END_VAR
VAR CONSTANT
	(* prefix to unify the test names *)
	TEST_NAME_PREFIX		:STRING := 'assert.dateAndTime.simple.dateAndTime.';
	(* max value of a DWORD *)
	{attribute 'hide'}
	MAX_DWORD				:DWORD := 16#FFFF_FFFF;
	(* min value of a DWORD *)
	{attribute 'hide'}
	MIN_DWORD				:DWORD := 16#0000_0000;
	(* only the msb is set *)
	{attribute 'hide'}
	MSB_ONLY				:DWORD := 16#8000_0000;
	(* only the msb is set *)
	{attribute 'hide'}
	LSB_ONLY				:DWORD := 16#0000_0001;
	(* all bits set except the msb *)
	{attribute 'hide'}
	WITHOUT_MSB 			:DWORD := 16#7FFF_FFFF;
	(* for every nibble is the msb set only *)
	{attribute 'hide'}
	ALL_NIBBLE_MSB			:DWORD := 16#8888_8888;
	(* for every nibble is the msb unset only *)
	{attribute 'hide'}
	WITHOUT_NIBBLE_MSB		:DWORD := 16#7777_7777;
	(* for every nibble is the lsb set only *)
	{attribute 'hide'}
	ALL_NIBBLE_LSB			:DWORD := 16#1111_1111;
	(* every bit is set except the lsb *)
	{attribute 'hide'}
	LSB_IS_UNSET			:DWORD := 16#FFFF_FFFE;
	(* max vale of date and time *)
	DT_MAX					:DT := TO_DT(MAX_DWORD);
	(* min vale of date and time *)
	DT_MIN					:DT := TO_DT(MIN_DWORD);
	(* only the msb is set *)
	DT_MSB_ONLY				:DT := TO_DT(MSB_ONLY);
	(* all bits set except the msb *)
	DT_WITHOUT_MSB 			:DT := TO_DT(WITHOUT_MSB);
	(* for every nibble is the msb set only *)
	DT_ALL_NIBBLE_MSB		:DT := TO_DT(ALL_NIBBLE_MSB);
	(* for every nibble is the msb unset only *)
	DT_WITHOUT_NIBBLE_MSB	:DT := TO_DT(WITHOUT_NIBBLE_MSB);
	(* for every nibble is the lsb set only *)
	DT_ALL_NIBBLE_LSB		:DT := TO_DT(ALL_NIBBLE_LSB);	
	(* every bit is set except the lsb *)
	DT_LSB_IS_UNSET			:DT := TO_DT(LSB_IS_UNSET);
	(* only the msb is set *)
	DT_LSB_ONLY				:DT := TO_DT(LSB_ONLY);
END_VAR

THIS^.runValueIsEqualToTests();
THIS^.runValueIsGreaterThanTests();
THIS^.runValueIsInRangeOfTests();
THIS^.runValueIsLessThanTests();
THIS^.runValueIsMaxTests();
THIS^.runValueIsMinTests();
THIS^.runValueIsNotEqualToTests();

(*

short summary
==================
This test method is a helper function to create a unified test name

.. <legal notes>

legal notes
=================
| SPDX-FileCopyrightText: © 2022 ekvip automation GmbH <info@ekvip.de>
| SPDX-License-Identifier: Apache-2.0
| For details check: Apache-2.0_

.. _Apache-2.0: https://www.apache.org/licenses/LICENSE-2.0

.. </legal notes>

parameters
==========

*)

METHOD PROTECTED getTestNameFor :Tc2_System.T_MaxString
VAR_INPUT
	(* name of the method to test, to create a unified test name *)
	nameOfMethodToTest	:Tc2_System.T_MaxString;
END_VAR
getTestNameFor := Tc2_Standard.CONCAT(THIS^.TEST_NAME_PREFIX, nameOfMethodToTest);
END_METHOD

(*

short summary
==================
This test method tests ``assert.dateAndTime.simple.dateAndTime.valueIsEqualTo``
method of CNM_AssertionInterfaceLib library with various inputs

.. <legal notes>

legal notes
=================
| SPDX-FileCopyrightText: © 2022 ekvip automation GmbH <info@ekvip.de>
| SPDX-License-Identifier: Apache-2.0
| For details check: Apache-2.0_

.. _Apache-2.0: https://www.apache.org/licenses/LICENSE-2.0

.. </legal notes>

*)

METHOD runValueIsEqualToTests
RETURN (NOT TcUnit.TEST_ORDERED(THIS^.getTestNameFor('valueIsEqualTo')));

THIS^.testValueIsEqualTo(
	valueToTest := THIS^.DT_MAX,
	expected := THIS^.DT_MAX
);
THIS^.testValueIsEqualTo(
	valueToTest := THIS^.DT_MIN,
	expected := THIS^.DT_MIN
);
THIS^.testValueIsEqualTo(
	valueToTest := THIS^.DT_MIN,
	expected := THIS^.DT_MAX
);
THIS^.testValueIsEqualTo(
	valueToTest := THIS^.DT_MAX,
	expected := THIS^.DT_MIN
);
THIS^.testValueIsEqualTo(
	valueToTest := THIS^.DT_ALL_NIBBLE_LSB,
	expected := THIS^.DT_ALL_NIBBLE_LSB
);
THIS^.testValueIsEqualTo(
	valueToTest := THIS^.DT_LSB_ONLY,
	expected := THIS^.DT_MSB_ONLY
);
THIS^.testValueIsEqualTo(
	valueToTest := THIS^.DT_MSB_ONLY,
	expected := THIS^.DT_MSB_ONLY
);
THIS^.testValueIsEqualTo(
	valueToTest := THIS^.DT_MSB_ONLY,
	expected := THIS^.DT_LSB_ONLY
);

TcUnit.TEST_FINISHED();
END_METHOD

(*

short summary
==================
This test method tests ``assert.dateAndTime.simple.dateAndTime.valueIsGreaterThan``
method of CNM_AssertionInterfaceLib library with various inputs

.. <legal notes>

legal notes
=================
| SPDX-FileCopyrightText: © 2022 ekvip automation GmbH <info@ekvip.de>
| SPDX-License-Identifier: Apache-2.0
| For details check: Apache-2.0_

.. _Apache-2.0: https://www.apache.org/licenses/LICENSE-2.0

.. </legal notes>

*)

METHOD runValueIsGreaterThanTests
RETURN (NOT TcUnit.TEST_ORDERED(THIS^.getTestNameFor('valueIsGreaterThan')));

THIS^.testValueIsGreaterThan(
	valueToTest := THIS^.DT_MAX,
	lessValue := THIS^.DT_MAX
);
THIS^.testValueIsGreaterThan(
	valueToTest := THIS^.DT_MIN,
	lessValue := THIS^.DT_MIN
);
THIS^.testValueIsGreaterThan(
	valueToTest := THIS^.DT_MIN,
	lessValue := THIS^.DT_MAX
);
THIS^.testValueIsGreaterThan(
	valueToTest := THIS^.DT_MAX,
	lessValue := THIS^.DT_MIN
);
THIS^.testValueIsGreaterThan(
	valueToTest := THIS^.DT_ALL_NIBBLE_LSB,
	lessValue := THIS^.DT_ALL_NIBBLE_LSB
);
THIS^.testValueIsGreaterThan(
	valueToTest := THIS^.DT_ALL_NIBBLE_MSB,
	lessValue := THIS^.DT_ALL_NIBBLE_LSB
);
THIS^.testValueIsGreaterThan(
	valueToTest := THIS^.DT_ALL_NIBBLE_LSB,
	lessValue := THIS^.DT_ALL_NIBBLE_MSB
);
THIS^.testValueIsGreaterThan(
	valueToTest := THIS^.DT_LSB_ONLY,
	lessValue := THIS^.DT_MSB_ONLY
);
THIS^.testValueIsGreaterThan(
	valueToTest := THIS^.DT_MSB_ONLY,
	lessValue := THIS^.DT_MSB_ONLY
);
THIS^.testValueIsGreaterThan(
	valueToTest := THIS^.DT_MSB_ONLY,
	lessValue := THIS^.DT_LSB_ONLY
);
THIS^.testValueIsGreaterThan(
	valueToTest := THIS^.DT_LSB_IS_UNSET,
	lessValue := THIS^.DT_MAX
);
THIS^.testValueIsGreaterThan(
	valueToTest := THIS^.DT_MAX,
	lessValue := THIS^.DT_LSB_IS_UNSET
);
TcUnit.TEST_FINISHED();
END_METHOD

(*

short summary
==================
This test method tests ``assert.dateAndTime.simple.dateAndTime.valueIsInRangeOf``
method of CNM_AssertionInterfaceLib library with various inputs

.. <legal notes>

legal notes
=================
| SPDX-FileCopyrightText: © 2022 ekvip automation GmbH <info@ekvip.de>
| SPDX-License-Identifier: Apache-2.0
| For details check: Apache-2.0_

.. _Apache-2.0: https://www.apache.org/licenses/LICENSE-2.0

.. </legal notes>

*)

METHOD runValueIsInRangeOfTests
RETURN (NOT TcUnit.TEST_ORDERED(THIS^.getTestNameFor('valueIsInRangeOf')));

THIS^.testValueIsInRangeOf(
	lowerLimit := THIS^.DT_MIN,
	valueToTest := THIS^.DT_MAX,
	upperLimit	:= THIS^.DT_MAX
);
THIS^.testValueIsInRangeOf(
	lowerLimit := THIS^.DT_MIN,
	valueToTest := THIS^.DT_MIN,
	upperLimit	:= THIS^.DT_MAX
);
THIS^.testValueIsInRangeOf(
	lowerLimit := THIS^.DT_MAX,
	valueToTest := THIS^.DT_MAX,
	upperLimit	:= THIS^.DT_MIN
);
THIS^.testValueIsInRangeOf(
	lowerLimit := THIS^.DT_MAX,
	valueToTest := THIS^.DT_MIN,
	upperLimit	:= THIS^.DT_MIN
);
THIS^.testValueIsInRangeOf(
	lowerLimit := THIS^.DT_LSB_IS_UNSET,
	valueToTest := THIS^.DT_MIN,
	upperLimit	:= THIS^.DT_MAX
);
THIS^.testValueIsInRangeOf(
	lowerLimit := THIS^.DT_MIN,
	valueToTest := THIS^.DT_LSB_IS_UNSET,
	upperLimit	:= THIS^.DT_MAX
);
THIS^.testValueIsInRangeOf(
	lowerLimit := THIS^.DT_LSB_IS_UNSET,
	valueToTest := THIS^.DT_LSB_IS_UNSET,
	upperLimit	:= THIS^.DT_LSB_IS_UNSET
);
THIS^.testValueIsInRangeOf(
	lowerLimit := THIS^.DT_ALL_NIBBLE_LSB,
	valueToTest := THIS^.DT_LSB_IS_UNSET,
	upperLimit	:= THIS^.DT_ALL_NIBBLE_MSB
);
THIS^.testValueIsInRangeOf(
	lowerLimit := THIS^.DT_LSB_IS_UNSET,
	valueToTest := THIS^.DT_ALL_NIBBLE_LSB,
	upperLimit	:= THIS^.DT_ALL_NIBBLE_MSB
);
THIS^.testValueIsInRangeOf(
	lowerLimit := THIS^.DT_LSB_ONLY,
	valueToTest := THIS^.DT_WITHOUT_MSB,
	upperLimit	:= THIS^.DT_MSB_ONLY
);
THIS^.testValueIsInRangeOf(
	lowerLimit := THIS^.DT_WITHOUT_MSB,
	valueToTest := THIS^.DT_LSB_ONLY,
	upperLimit	:= THIS^.DT_MSB_ONLY
);
THIS^.testValueIsInRangeOf(
	lowerLimit := THIS^.DT_WITHOUT_NIBBLE_MSB,
	valueToTest := THIS^.DT_MAX,
	upperLimit	:= THIS^.DT_ALL_NIBBLE_MSB
);
THIS^.testValueIsInRangeOf(
	lowerLimit := THIS^.DT_WITHOUT_NIBBLE_MSB,
	valueToTest := THIS^.DT_MIN,
	upperLimit	:= THIS^.DT_ALL_NIBBLE_MSB
);
THIS^.testValueIsInRangeOf(
	lowerLimit := THIS^.DT_WITHOUT_NIBBLE_MSB,
	valueToTest := THIS^.DT_WITHOUT_NIBBLE_MSB,
	upperLimit	:= THIS^.DT_ALL_NIBBLE_MSB
);
THIS^.testValueIsInRangeOf(
	lowerLimit := THIS^.DT_WITHOUT_NIBBLE_MSB,
	valueToTest := THIS^.DT_ALL_NIBBLE_MSB,
	upperLimit	:= THIS^.DT_ALL_NIBBLE_MSB
);
TcUnit.TEST_FINISHED();
END_METHOD

(*

short summary
==================
This test method tests ``assert.dateAndTime.simple.dateAndTime.valueIsLessThan``
method of CNM_AssertionInterfaceLib library with various inputs

.. <legal notes>

legal notes
=================
| SPDX-FileCopyrightText: © 2022 ekvip automation GmbH <info@ekvip.de>
| SPDX-License-Identifier: Apache-2.0
| For details check: Apache-2.0_

.. _Apache-2.0: https://www.apache.org/licenses/LICENSE-2.0

.. </legal notes>

*)

METHOD runValueIsLessThanTests
RETURN (NOT TcUnit.TEST_ORDERED(THIS^.getTestNameFor('valueIsLessThan')));

THIS^.testValueIsLessThan(
	valueToTest := THIS^.DT_MAX,
	greaterValue := THIS^.DT_MAX
);
THIS^.testValueIsLessThan(
	valueToTest := THIS^.DT_MIN,
	greaterValue := THIS^.DT_MIN
);
THIS^.testValueIsLessThan(
	valueToTest := THIS^.DT_MIN,
	greaterValue := THIS^.DT_MAX
);
THIS^.testValueIsLessThan(
	valueToTest := THIS^.DT_MAX,
	greaterValue := THIS^.DT_MIN
);
THIS^.testValueIsLessThan(
	valueToTest := THIS^.DT_ALL_NIBBLE_LSB,
	greaterValue := THIS^.DT_ALL_NIBBLE_LSB
);
THIS^.testValueIsLessThan(
	valueToTest := THIS^.DT_ALL_NIBBLE_MSB,
	greaterValue := THIS^.DT_ALL_NIBBLE_LSB
);
THIS^.testValueIsLessThan(
	valueToTest := THIS^.DT_ALL_NIBBLE_LSB,
	greaterValue := THIS^.DT_ALL_NIBBLE_MSB
);
THIS^.testValueIsLessThan(
	valueToTest := THIS^.DT_LSB_ONLY,
	greaterValue := THIS^.DT_MSB_ONLY
);
THIS^.testValueIsLessThan(
	valueToTest := THIS^.DT_MSB_ONLY,
	greaterValue := THIS^.DT_MSB_ONLY
);
THIS^.testValueIsLessThan(
	valueToTest := THIS^.DT_MSB_ONLY,
	greaterValue := THIS^.DT_LSB_ONLY
);
THIS^.testValueIsLessThan(
	valueToTest := THIS^.DT_LSB_IS_UNSET,
	greaterValue := THIS^.DT_MAX
);
THIS^.testValueIsLessThan(
	valueToTest := THIS^.DT_MAX,
	greaterValue := THIS^.DT_LSB_IS_UNSET
);
TcUnit.TEST_FINISHED();
END_METHOD

(*

short summary
==================
This test method tests ``assert.dateAndTime.simple.dateAndTime.valueIsMax``
method of CNM_AssertionInterfaceLib library with various inputs

.. <legal notes>

legal notes
=================
| SPDX-FileCopyrightText: © 2022 ekvip automation GmbH <info@ekvip.de>
| SPDX-License-Identifier: Apache-2.0
| For details check: Apache-2.0_

.. _Apache-2.0: https://www.apache.org/licenses/LICENSE-2.0

.. </legal notes>

*)

METHOD runValueIsMaxTests
RETURN (NOT TcUnit.TEST_ORDERED(THIS^.getTestNameFor('valueIsMax')));

THIS^.testValueIsMax(
	valueToTest := THIS^.DT_MAX,
	maximumValue := THIS^.DT_MAX
);
THIS^.testValueIsMax(
	valueToTest := THIS^.DT_MIN,
	maximumValue := THIS^.DT_MIN
);
THIS^.testValueIsMax(
	valueToTest := THIS^.DT_MIN,
	maximumValue := THIS^.DT_MAX
);
THIS^.testValueIsMax(
	valueToTest := THIS^.DT_MAX,
	maximumValue := THIS^.DT_MIN
);
THIS^.testValueIsMax(
	valueToTest := THIS^.DT_ALL_NIBBLE_LSB,
	maximumValue := THIS^.DT_ALL_NIBBLE_LSB
);
THIS^.testValueIsMax(
	valueToTest := THIS^.DT_ALL_NIBBLE_MSB,
	maximumValue := THIS^.DT_ALL_NIBBLE_LSB
);
THIS^.testValueIsMax(
	valueToTest := THIS^.DT_ALL_NIBBLE_LSB,
	maximumValue := THIS^.DT_ALL_NIBBLE_MSB
);
THIS^.testValueIsMax(
	valueToTest := THIS^.DT_LSB_ONLY,
	maximumValue := THIS^.DT_MSB_ONLY
);
THIS^.testValueIsMax(
	valueToTest := THIS^.DT_MSB_ONLY,
	maximumValue := THIS^.DT_MSB_ONLY
);
THIS^.testValueIsMax(
	valueToTest := THIS^.DT_MSB_ONLY,
	maximumValue := THIS^.DT_LSB_ONLY
);
THIS^.testValueIsMax(
	valueToTest := THIS^.DT_LSB_IS_UNSET,
	maximumValue := THIS^.DT_MAX
);
THIS^.testValueIsMax(
	valueToTest := THIS^.DT_MAX,
	maximumValue := THIS^.DT_LSB_IS_UNSET
);
TcUnit.TEST_FINISHED();
END_METHOD

(*

short summary
==================
This test method tests ``assert.dateAndTime.simple.dateAndTime.valueIsMin``
method of CNM_AssertionInterfaceLib library with various inputs

.. <legal notes>

legal notes
=================
| SPDX-FileCopyrightText: © 2022 ekvip automation GmbH <info@ekvip.de>
| SPDX-License-Identifier: Apache-2.0
| For details check: Apache-2.0_

.. _Apache-2.0: https://www.apache.org/licenses/LICENSE-2.0

.. </legal notes>

*)

METHOD runValueIsMinTests
RETURN (NOT TcUnit.TEST_ORDERED(THIS^.getTestNameFor('valueIsMin')));

THIS^.testValueIsMin(
	valueToTest := THIS^.DT_MAX,
	minimumValue := THIS^.DT_MAX
);
THIS^.testValueIsMin(
	valueToTest := THIS^.DT_MIN,
	minimumValue := THIS^.DT_MIN
);
THIS^.testValueIsMin(
	valueToTest := THIS^.DT_MIN,
	minimumValue := THIS^.DT_MAX
);
THIS^.testValueIsMin(
	valueToTest := THIS^.DT_MAX,
	minimumValue := THIS^.DT_MIN
);
THIS^.testValueIsMin(
	valueToTest := THIS^.DT_ALL_NIBBLE_LSB,
	minimumValue := THIS^.DT_ALL_NIBBLE_LSB
);
THIS^.testValueIsMin(
	valueToTest := THIS^.DT_ALL_NIBBLE_MSB,
	minimumValue := THIS^.DT_ALL_NIBBLE_LSB
);
THIS^.testValueIsMin(
	valueToTest := THIS^.DT_ALL_NIBBLE_LSB,
	minimumValue := THIS^.DT_ALL_NIBBLE_MSB
);
THIS^.testValueIsMin(
	valueToTest := THIS^.DT_LSB_ONLY,
	minimumValue := THIS^.DT_MSB_ONLY
);
THIS^.testValueIsMin(
	valueToTest := THIS^.DT_MSB_ONLY,
	minimumValue := THIS^.DT_MSB_ONLY
);
THIS^.testValueIsMin(
	valueToTest := THIS^.DT_MSB_ONLY,
	minimumValue := THIS^.DT_LSB_ONLY
);
THIS^.testValueIsMin(
	valueToTest := THIS^.DT_LSB_IS_UNSET,
	minimumValue := THIS^.DT_MAX
);
THIS^.testValueIsMin(
	valueToTest := THIS^.DT_MAX,
	minimumValue := THIS^.DT_LSB_IS_UNSET
);
TcUnit.TEST_FINISHED();
END_METHOD

(*

short summary
==================
This test method tests ``assert.dateAndTime.simple.dateAndTime.valueIsNotEqualTo``
method of CNM_AssertionInterfaceLib library with various inputs

.. <legal notes>

legal notes
=================
| SPDX-FileCopyrightText: © 2022 ekvip automation GmbH <info@ekvip.de>
| SPDX-License-Identifier: Apache-2.0
| For details check: Apache-2.0_

.. _Apache-2.0: https://www.apache.org/licenses/LICENSE-2.0

.. </legal notes>

*)

METHOD runValueIsNotEqualToTests
RETURN (NOT TcUnit.TEST_ORDERED(THIS^.getTestNameFor('valueIsNotEqualTo')));

THIS^.testValueIsNotEqualTo(
	valueToTest := THIS^.DT_MAX,
	unexpectedValue := THIS^.DT_MAX
);
THIS^.testValueIsNotEqualTo(
	valueToTest := THIS^.DT_MIN,
	unexpectedValue := THIS^.DT_MIN
);
THIS^.testValueIsNotEqualTo(
	valueToTest := THIS^.DT_MIN,
	unexpectedValue := THIS^.DT_MAX
);
THIS^.testValueIsNotEqualTo(
	valueToTest := THIS^.DT_MAX,
	unexpectedValue := THIS^.DT_MIN
);
THIS^.testValueIsNotEqualTo(
	valueToTest := THIS^.DT_ALL_NIBBLE_LSB,
	unexpectedValue := THIS^.DT_ALL_NIBBLE_LSB
);
THIS^.testValueIsNotEqualTo(
	valueToTest := THIS^.DT_LSB_ONLY,
	unexpectedValue := THIS^.DT_MSB_ONLY
);
THIS^.testValueIsNotEqualTo(
	valueToTest := THIS^.DT_MSB_ONLY,
	unexpectedValue := THIS^.DT_MSB_ONLY
);
THIS^.testValueIsNotEqualTo(
	valueToTest := THIS^.DT_MSB_ONLY,
	unexpectedValue := THIS^.DT_LSB_ONLY
);

TcUnit.TEST_FINISHED();
END_METHOD

(*

short summary
==================
This test method tests ``assert.dateAndTime.simple.dateAndTime.valueIsEqualTo``
method of CNM_AssertionInterfaceLib library, 
it provides the possibility to handover test data via parameter 


.. <legal notes>

legal notes
=================
| SPDX-FileCopyrightText: © 2022 ekvip automation GmbH <info@ekvip.de>
| SPDX-License-Identifier: Apache-2.0
| For details check: Apache-2.0_

.. _Apache-2.0: https://www.apache.org/licenses/LICENSE-2.0

.. </legal notes>

parameters
==========

*)

METHOD testValueIsEqualTo 
VAR_INPUT
	(* for the test it's the parameter ``currentValue`` *)
	valueToTest	:DT;
	(* for the test it's the parameter ``expectedValue`` *)
	expected	:DT;
END_VAR
VAR
	(* just the expectation if the assertion to test must be worng or true *)
	assertionIsWrong		:BOOL;
	(* contains the format string for the test message *)
	message					:Tc2_System.T_MaxString;
	(* TwinCAT printf with the test message *)
	messageStringBuilder	:Tc2_Utilities.FB_FormatString;
	(* dt value of ``currentValue`` as string *)
	currentValueAsString	:STRING(22);
	(* dt value of ``expectedValue`` as string *)
	expectedValueAsString	:STRING(22);
END_VAR
THIS^.assertorContainer.resetAssertor();

assertionIsWrong := (valueToTest <> expected);
message := SEL(
	assertionIsWrong,
	'currentValue is %s expectedValue is %s assertion must be TRUE', 
	'currentValue is %s expectedValue is %s assertion must be FALSE'
);
currentValueAsString := TO_STRING(valueToTest);
expectedValueAsString := TO_STRING(expected);

messageStringBuilder(
	sFormat := message,
	arg1 := THIS^.AnyToArg(currentValueAsString),
	arg2 := THIS^.AnyToArg(expectedValueAsString)
);

THIS^.assertorContainer.assertor.assert.dateAndTime.simple.dateAndTime.valueIsEqualTo(
	currentValue	:= valueToTest,
	expectedValue	:= expected,
	message			:= ''
   );

THIS^.AssertEquals_BOOL(
	Expected 	:= assertionIsWrong,
	Actual 		:= THIS^.assertorContainer.wasAssertionWrong,
	Message 	:= messageStringBuilder.sOut
);
END_METHOD

(*

short summary
==================
This test method tests ``assert.dateAndTime.simple.dateAndTime.valueIsGreaterThan``
method of CNM_AssertionInterfaceLib library, 
it provides the possibility to handover test data via parameter 


.. <legal notes>

legal notes
=================
| SPDX-FileCopyrightText: © 2022 ekvip automation GmbH <info@ekvip.de>
| SPDX-License-Identifier: Apache-2.0
| For details check: Apache-2.0_

.. _Apache-2.0: https://www.apache.org/licenses/LICENSE-2.0

.. </legal notes>

parameters
==========

*)

METHOD testValueIsGreaterThan 
VAR_INPUT
	(* for the test it's the parameter ``currentValue`` *)
	valueToTest	:DT;
	(* for the test it's the parameter ``lessValue`` *)
	lessValue	:DT;
END_VAR
VAR
	(* just the expectation if the assertion to test must be worng or true *)
	assertionIsWrong		:BOOL;
	(* contains the format string for the test message *)
	message					:Tc2_System.T_MaxString;
	(* TwinCAT printf with the test message *)
	messageStringBuilder	:Tc2_Utilities.FB_FormatString;
	(* dt value of ``currentValue`` as string *)
	currentValueAsString	:STRING(22);
	(* dt value of ``lessValue`` as string *)
	lessValueAsString		:STRING(22);
END_VAR
THIS^.assertorContainer.resetAssertor();

assertionIsWrong := (valueToTest <= lessValue);
message := SEL(
	assertionIsWrong,
	'currentValue is %s lessValue is %s assertion must be TRUE', 
	'currentValue is %s lessValue is %s assertion must be FALSE'
);
currentValueAsString := TO_STRING(valueToTest);
lessValueAsString := TO_STRING(lessValue);

messageStringBuilder(
	sFormat := message,
	arg1 := THIS^.AnyToArg(currentValueAsString),
	arg2 := THIS^.AnyToArg(lessValueAsString)
);

THIS^.assertorContainer.assertor.assert.dateAndTime.simple.dateAndTime.valueIsGreaterThan(
	currentValue	:= valueToTest,
	lessValue		:= lessValue,
	message			:= ''
   );

THIS^.AssertEquals_BOOL(
	Expected 	:= assertionIsWrong,
	Actual 		:= THIS^.assertorContainer.wasAssertionWrong,
	Message 	:= messageStringBuilder.sOut
);
END_METHOD

(*

short summary
==================
This test method tests ``assert.dateAndTime.simple.dateAndTime.valueIsInRangeOf``
method of CNM_AssertionInterfaceLib library, 
it provides the possibility to handover test data via parameter 


.. <legal notes>

legal notes
=================
| SPDX-FileCopyrightText: © 2022 ekvip automation GmbH <info@ekvip.de>
| SPDX-License-Identifier: Apache-2.0
| For details check: Apache-2.0_

.. _Apache-2.0: https://www.apache.org/licenses/LICENSE-2.0

.. </legal notes>

parameters
==========

*)

METHOD testValueIsInRangeOf 
VAR_INPUT
	(* for the test it's the parameter ``lowerLimit`` *)
	lowerLimit	:DT;
	(* for the test it's the parameter ``currentValue`` *)
	valueToTest	:DT;
	(* for the test it's the parameter ``upperLimit`` *)
	upperLimit	:DT;
END_VAR
VAR
	(* just the expectation if the assertion to test must be worng or true *)
	assertionIsWrong		:BOOL;
	(* contains the format string for the test message *)
	message					:Tc2_System.T_MaxString;
	(* TwinCAT printf with the test message *)
	messageStringBuilder	:Tc2_Utilities.FB_FormatString;
	(* dt value of ``lowerLimit`` as string *)
	lowerLimitAsString		:STRING(22);
	(* dt value of ``currentValue`` as string *)
	currentValueAsString	:STRING(22);
	(* dt value of ``upperLimit`` as string *)
	upperLimitAsString		:STRING(22);

END_VAR
THIS^.assertorContainer.resetAssertor();

assertionIsWrong := ((valueToTest < lowerLimit) OR (valueToTest > upperLimit));
message := SEL(
	assertionIsWrong,
	'lowerLimit is %s currentValue is %s upperLimit is %s assertion must be TRUE', 
	'lowerLimit is %s currentValue is %s upperLimit is %s assertion must be FALSE'
);
lowerLimitAsString		:= TO_STRING(lowerLimit);
currentValueAsString	:= TO_STRING(valueToTest);
upperLimitAsString		:= TO_STRING(upperLimit);

messageStringBuilder(
	sFormat := message,
	arg1 := THIS^.AnyToArg(lowerLimitAsString),
	arg2 := THIS^.AnyToArg(currentValueAsString),
	arg3 := THIS^.AnyToArg(upperLimitAsString)
);

THIS^.assertorContainer.assertor.assert.dateAndTime.simple.dateAndTime.valueIsInRangeOf(
	lowerLimit		:= lowerLimit,
	currentValue	:= valueToTest,
	upperLimit		:= upperLimit,
	message			:= ''
   );

THIS^.AssertEquals_BOOL(
	Expected 	:= assertionIsWrong,
	Actual 		:= THIS^.assertorContainer.wasAssertionWrong,
	Message 	:= messageStringBuilder.sOut
);
END_METHOD

(*

short summary
==================
This test method tests ``assert.dateAndTime.simple.dateAndTime.valueIsLessThan``
method of CNM_AssertionInterfaceLib library, 
it provides the possibility to handover test data via parameter 


.. <legal notes>

legal notes
=================
| SPDX-FileCopyrightText: © 2022 ekvip automation GmbH <info@ekvip.de>
| SPDX-License-Identifier: Apache-2.0
| For details check: Apache-2.0_

.. _Apache-2.0: https://www.apache.org/licenses/LICENSE-2.0

.. </legal notes>

parameters
==========

*)

METHOD testValueIsLessThan 
VAR_INPUT
	(* for the test it's the parameter ``currentValue`` *)
	valueToTest		:DT;
	(* for the test it's the parameter ``greaterValue`` *)
	greaterValue	:DT;
END_VAR
VAR
	(* just the expectation if the assertion to test must be worng or true *)
	assertionIsWrong		:BOOL;
	(* contains the format string for the test message *)
	message					:Tc2_System.T_MaxString;
	(* TwinCAT printf with the test message *)
	messageStringBuilder	:Tc2_Utilities.FB_FormatString;
	(* dt value of ``currentValue`` as string *)
	currentValueAsString	:STRING(22);
	(* dt value of ``greaterValue`` as string *)
	greaterValueAsString	:STRING(22);
END_VAR
THIS^.assertorContainer.resetAssertor();

assertionIsWrong := (valueToTest >= greaterValue);
message := SEL(
	assertionIsWrong,
	'currentValue is %s greaterValue is %s assertion must be TRUE', 
	'currentValue is %s greaterValue is %s assertion must be FALSE'
);
currentValueAsString := TO_STRING(valueToTest);
greaterValueAsString := TO_STRING(greaterValue);

messageStringBuilder(
	sFormat := message,
	arg1 := THIS^.AnyToArg(currentValueAsString),
	arg2 := THIS^.AnyToArg(greaterValueAsString)
);

THIS^.assertorContainer.assertor.assert.dateAndTime.simple.dateAndTime.valueIsLessThan(
	currentValue	:= valueToTest,
	greaterValue	:= greaterValue,
	message			:= ''
   );

THIS^.AssertEquals_BOOL(
	Expected 	:= assertionIsWrong,
	Actual 		:= THIS^.assertorContainer.wasAssertionWrong,
	Message 	:= messageStringBuilder.sOut
);
END_METHOD

(*

short summary
==================
This test method tests ``assert.dateAndTime.simple.dateAndTime.valueIsMax``
method of CNM_AssertionInterfaceLib library, 
it provides the possibility to handover test data via parameter 


.. <legal notes>

legal notes
=================
| SPDX-FileCopyrightText: © 2022 ekvip automation GmbH <info@ekvip.de>
| SPDX-License-Identifier: Apache-2.0
| For details check: Apache-2.0_

.. _Apache-2.0: https://www.apache.org/licenses/LICENSE-2.0

.. </legal notes>

parameters
==========

*)

METHOD testValueIsMax 
VAR_INPUT
	(* for the test it's the parameter ``currentValue`` *)
	valueToTest		:DT;
	(* for the test it's the parameter ``greaterValue`` *)
	maximumValue	:DT;
END_VAR
VAR
	(* just the expectation if the assertion to test must be worng or true *)
	assertionIsWrong		:BOOL;
	(* contains the format string for the test message *)
	message					:Tc2_System.T_MaxString;
	(* TwinCAT printf with the test message *)
	messageStringBuilder	:Tc2_Utilities.FB_FormatString;
	(* dt value of ``currentValue`` as string *)
	currentValueAsString	:STRING(22);
	(* dt value of ``maximumValue`` as string *)
	maximumValueAsString	:STRING(22);
END_VAR
THIS^.assertorContainer.resetAssertor();

assertionIsWrong := (valueToTest > maximumValue);
message := SEL(
	assertionIsWrong,
	'currentValue is %s maximumValue is %s assertion must be TRUE', 
	'currentValue is %s maximumValue is %s assertion must be FALSE'
);
currentValueAsString := TO_STRING(valueToTest);
maximumValueAsString := TO_STRING(maximumValue);

messageStringBuilder(
	sFormat := message,
	arg1 := THIS^.AnyToArg(currentValueAsString),
	arg2 := THIS^.AnyToArg(maximumValueAsString)
);

THIS^.assertorContainer.assertor.assert.dateAndTime.simple.dateAndTime.valueIsMax(
	currentValue	:= valueToTest,
	maximumValue	:= maximumValue,
	message			:= ''
   );

THIS^.AssertEquals_BOOL(
	Expected 	:= assertionIsWrong,
	Actual 		:= THIS^.assertorContainer.wasAssertionWrong,
	Message 	:= messageStringBuilder.sOut
);
END_METHOD

(*

short summary
==================
This test method tests ``assert.dateAndTime.simple.dateAndTime.valueIsMin``
method of CNM_AssertionInterfaceLib library, 
it provides the possibility to handover test data via parameter 


.. <legal notes>

legal notes
=================
| SPDX-FileCopyrightText: © 2022 ekvip automation GmbH <info@ekvip.de>
| SPDX-License-Identifier: Apache-2.0
| For details check: Apache-2.0_

.. _Apache-2.0: https://www.apache.org/licenses/LICENSE-2.0

.. </legal notes>

parameters
==========

*)

METHOD testValueIsMin 
VAR_INPUT
	(* for the test it's the parameter ``currentValue`` *)
	valueToTest		:DT;
	(* for the test it's the parameter ``greaterValue`` *)
	minimumValue	:DT;
END_VAR
VAR
	(* just the expectation if the assertion to test must be worng or true *)
	assertionIsWrong		:BOOL;
	(* contains the format string for the test message *)
	message					:Tc2_System.T_MaxString;
	(* TwinCAT printf with the test message *)
	messageStringBuilder	:Tc2_Utilities.FB_FormatString;
	(* dt value of ``currentValue`` as string *)
	currentValueAsString	:STRING(22);
	(* dt value of ``minimumValue`` as string *)
	minimumValueAsString	:STRING(22);
END_VAR
THIS^.assertorContainer.resetAssertor();

assertionIsWrong := (valueToTest < minimumValue);
message := SEL(
	assertionIsWrong,
	'currentValue is %s minimumValue is %s assertion must be TRUE', 
	'currentValue is %s minimumValue is %s assertion must be FALSE'
);
currentValueAsString := TO_STRING(valueToTest);
minimumValueAsString := TO_STRING(minimumValue);

messageStringBuilder(
	sFormat := message,
	arg1 := THIS^.AnyToArg(currentValueAsString),
	arg2 := THIS^.AnyToArg(minimumValueAsString)
);

THIS^.assertorContainer.assertor.assert.dateAndTime.simple.dateAndTime.valueIsMin(
	currentValue	:= valueToTest,
	minimumValue	:= minimumValue,
	message			:= ''
   );

THIS^.AssertEquals_BOOL(
	Expected 	:= assertionIsWrong,
	Actual 		:= THIS^.assertorContainer.wasAssertionWrong,
	Message 	:= messageStringBuilder.sOut
);
END_METHOD

(*

short summary
==================
This test method tests ``assert.dateAndTime.simple.dateAndTime.valueIsNotEqualTo``
method of CNM_AssertionInterfaceLib library, 
it provides the possibility to handover test data via parameter 


.. <legal notes>

legal notes
=================
| SPDX-FileCopyrightText: © 2022 ekvip automation GmbH <info@ekvip.de>
| SPDX-License-Identifier: Apache-2.0
| For details check: Apache-2.0_

.. _Apache-2.0: https://www.apache.org/licenses/LICENSE-2.0

.. </legal notes>

parameters
==========

*)

METHOD testValueIsNotEqualTo 
VAR_INPUT
	(* for the test it's the parameter ``currentValue`` *)
	valueToTest		:DT;
	(* for the test it's the parameter ``unexpectedValue`` *)
	unexpectedValue	:DT;
END_VAR
VAR
	(* just the expectation if the assertion to test must be worng or true *)
	assertionIsWrong		:BOOL;
	(* contains the format string for the test message *)
	message					:Tc2_System.T_MaxString;
	(* TwinCAT printf with the test message *)
	messageStringBuilder	:Tc2_Utilities.FB_FormatString;
	(* dt value of ``currentValue`` as string *)
	currentValueAsString	:STRING(22);
	(* dt value of ``unexpectedValue`` as string *)
	unexpectedValueAsString	:STRING(22);
END_VAR
THIS^.assertorContainer.resetAssertor();

assertionIsWrong := (valueToTest = unexpectedValue);
message := SEL(
	assertionIsWrong,
	'currentValue is %s expectedValue is %s assertion must be TRUE', 
	'currentValue is %s expectedValue is %s assertion must be FALSE'
);
currentValueAsString := TO_STRING(valueToTest);
unexpectedValueAsString := TO_STRING(unexpectedValue);

messageStringBuilder(
	sFormat := message,
	arg1 := THIS^.AnyToArg(currentValueAsString),
	arg2 := THIS^.AnyToArg(unexpectedValueAsString)
);

THIS^.assertorContainer.assertor.assert.dateAndTime.simple.dateAndTime.valueIsNotEqualTo(
	currentValue	:= valueToTest,
	unexpectedValue	:= unexpectedValue,
	message			:= ''
   );

THIS^.AssertEquals_BOOL(
	Expected 	:= assertionIsWrong,
	Actual 		:= THIS^.assertorContainer.wasAssertionWrong,
	Message 	:= messageStringBuilder.sOut
);
END_METHOD

END_FUNCTION_BLOCK

// ---- AssertionTester/AssertionTests/DateTimeAssertions/classes/DateAssertionTests.TcPOU
(*

short summary
==================
This class tests all methods of DATE assertions
with various combinations of inputs and checks expected 
outputs are satisfied or not

.. <legal notes>

legal notes
=================
| SPDX-FileCopyrightText: © 2022 ekvip automation GmbH <info@ekvip.de>
| SPDX-License-Identifier: Apache-2.0
| For details check: Apache-2.0_

.. _Apache-2.0: https://www.apache.org/licenses/LICENSE-2.0

.. </legal notes>

methods and properties
======================

*)


FUNCTION_BLOCK DateAssertionTests EXTENDS AbstractAssertorTest
VAR
	
END_VAR
VAR CONSTANT
	(* prefix to unify the test names *)
	TEST_NAME_PREFIX		:STRING := 'assert.dateAndTime.simple.dateOnly.';
	(* max value of a DWORD *)
	{attribute 'hide'}
	MAX_DWORD				:DWORD := 16#FFFF_FFFF;
	(* min value of a DWORD *)
	{attribute 'hide'}
	MIN_DWORD				:DWORD := 16#0000_0000;
	(* only the msb is set *)
	{attribute 'hide'}
	MSB_ONLY				:DWORD := 16#8000_0000;
	(* only the msb is set *)
	{attribute 'hide'}
	LSB_ONLY				:DWORD := 16#0000_0001;
	(* all bits set except the msb *)
	{attribute 'hide'}
	WITHOUT_MSB 			:DWORD := 16#7FFF_FFFF;
	(* for every nibble is the msb set only *)
	{attribute 'hide'}
	ALL_NIBBLE_MSB			:DWORD := 16#8888_8888;
	(* for every nibble is the msb unset only *)
	{attribute 'hide'}
	WITHOUT_NIBBLE_MSB		:DWORD := 16#7777_7777;
	(* for every nibble is the lsb set only *)
	{attribute 'hide'}
	ALL_NIBBLE_LSB			:DWORD := 16#1111_1111;
	(* every bit is set except the lsb *)
	{attribute 'hide'}
	LSB_IS_UNSET			:DWORD := 16#FFFF_FFFE;
	(* max vale of date and time *)
	DATE_MAX				:DATE := TO_DATE(MAX_DWORD);
	(* min vale of date and time *)
	DATE_MIN				:DATE := TO_DATE(MIN_DWORD);
	(* only the msb is set *)
	DATE_MSB_ONLY			:DATE := TO_DATE(MSB_ONLY);
	(* all bits set except the msb *)
	DATE_WITHOUT_MSB 		:DATE := TO_DATE(WITHOUT_MSB);
	(* for every nibble is the msb set only *)
	DATE_ALL_NIBBLE_MSB		:DATE := TO_DATE(ALL_NIBBLE_MSB);
	(* for every nibble is the msb unset only *)
	DATE_WITHOUT_NIBBLE_MSB	:DATE := TO_DATE(WITHOUT_NIBBLE_MSB);
	(* for every nibble is the lsb set only *)
	DATE_ALL_NIBBLE_LSB		:DATE := TO_DATE(ALL_NIBBLE_LSB);	
	(* every bit is set except the lsb *)
	DATE_LSB_IS_UNSET		:DATE := TO_DATE(LSB_IS_UNSET);
	(* only the msb is set *)
	DATE_LSB_ONLY			:DATE := TO_DATE(LSB_ONLY);
END_VAR

THIS^.runValueIsEqualToTests();
THIS^.runValueIsGreaterThanTests();
THIS^.runValueIsInRangeOfTests();
THIS^.runValueIsLessThanTests();
THIS^.runValueIsMaxTests();
THIS^.runValueIsMinTests();
THIS^.runValueIsNotEqualToTests();

(*

short summary
==================
This test method is a helper function to create a unified test name

.. <legal notes>

legal notes
=================
| SPDX-FileCopyrightText: © 2022 ekvip automation GmbH <info@ekvip.de>
| SPDX-License-Identifier: Apache-2.0
| For details check: Apache-2.0_

.. _Apache-2.0: https://www.apache.org/licenses/LICENSE-2.0

.. </legal notes>

parameters
==========

*)

METHOD PROTECTED getTestNameFor :Tc2_System.T_MaxString
VAR_INPUT
	(* name of the method to test, to create a unified test name *)
	nameOfMethodToTest	:Tc2_System.T_MaxString;
END_VAR
getTestNameFor := Tc2_Standard.CONCAT(THIS^.TEST_NAME_PREFIX, nameOfMethodToTest);
END_METHOD

(*

short summary
==================
This test method tests ``assert.dateAndTime.simple.dateOnly.valueIsEqualTo``
method of CNM_AssertionInterfaceLib library with various inputs

.. <legal notes>

legal notes
=================
| SPDX-FileCopyrightText: © 2022 ekvip automation GmbH <info@ekvip.de>
| SPDX-License-Identifier: Apache-2.0
| For details check: Apache-2.0_

.. _Apache-2.0: https://www.apache.org/licenses/LICENSE-2.0

.. </legal notes>

*)

METHOD runValueIsEqualToTests
RETURN (NOT TcUnit.TEST_ORDERED(THIS^.getTestNameFor('valueIsEqualTo')));

THIS^.testValueIsEqualTo(
	valueToTest := THIS^.DATE_MAX,
	expected := THIS^.DATE_MAX
);
THIS^.testValueIsEqualTo(
	valueToTest := THIS^.DATE_MIN,
	expected := THIS^.DATE_MIN
);
THIS^.testValueIsEqualTo(
	valueToTest := THIS^.DATE_MIN,
	expected := THIS^.DATE_MAX
);
THIS^.testValueIsEqualTo(
	valueToTest := THIS^.DATE_MAX,
	expected := THIS^.DATE_MIN
);
THIS^.testValueIsEqualTo(
	valueToTest := THIS^.DATE_ALL_NIBBLE_LSB,
	expected := THIS^.DATE_ALL_NIBBLE_LSB
);
THIS^.testValueIsEqualTo(
	valueToTest := THIS^.DATE_LSB_ONLY,
	expected := THIS^.DATE_MSB_ONLY
);
THIS^.testValueIsEqualTo(
	valueToTest := THIS^.DATE_MSB_ONLY,
	expected := THIS^.DATE_MSB_ONLY
);
THIS^.testValueIsEqualTo(
	valueToTest := THIS^.DATE_MSB_ONLY,
	expected := THIS^.DATE_LSB_ONLY
);

TcUnit.TEST_FINISHED();
END_METHOD

(*

short summary
==================
This test method tests ``assert.dateAndTime.simple.dateOnly.valueIsGreaterThan``
method of CNM_AssertionInterfaceLib library with various inputs

.. <legal notes>

legal notes
=================
| SPDX-FileCopyrightText: © 2022 ekvip automation GmbH <info@ekvip.de>
| SPDX-License-Identifier: Apache-2.0
| For details check: Apache-2.0_

.. _Apache-2.0: https://www.apache.org/licenses/LICENSE-2.0

.. </legal notes>

*)

METHOD runValueIsGreaterThanTests
RETURN (NOT TcUnit.TEST_ORDERED(THIS^.getTestNameFor('valueIsGreaterThan')));

THIS^.testValueIsGreaterThan(
	valueToTest := THIS^.DATE_MAX,
	lessValue := THIS^.DATE_MAX
);
THIS^.testValueIsGreaterThan(
	valueToTest := THIS^.DATE_MIN,
	lessValue := THIS^.DATE_MIN
);
THIS^.testValueIsGreaterThan(
	valueToTest := THIS^.DATE_MIN,
	lessValue := THIS^.DATE_MAX
);
THIS^.testValueIsGreaterThan(
	valueToTest := THIS^.DATE_MAX,
	lessValue := THIS^.DATE_MIN
);
THIS^.testValueIsGreaterThan(
	valueToTest := THIS^.DATE_ALL_NIBBLE_LSB,
	lessValue := THIS^.DATE_ALL_NIBBLE_LSB
);
THIS^.testValueIsGreaterThan(
	valueToTest := THIS^.DATE_ALL_NIBBLE_MSB,
	lessValue := THIS^.DATE_ALL_NIBBLE_LSB
);
THIS^.testValueIsGreaterThan(
	valueToTest := THIS^.DATE_ALL_NIBBLE_LSB,
	lessValue := THIS^.DATE_ALL_NIBBLE_MSB
);
THIS^.testValueIsGreaterThan(
	valueToTest := THIS^.DATE_LSB_ONLY,
	lessValue := THIS^.DATE_MSB_ONLY
);
THIS^.testValueIsGreaterThan(
	valueToTest := THIS^.DATE_MSB_ONLY,
	lessValue := THIS^.DATE_MSB_ONLY
);
THIS^.testValueIsGreaterThan(
	valueToTest := THIS^.DATE_MSB_ONLY,
	lessValue := THIS^.DATE_LSB_ONLY
);
THIS^.testValueIsGreaterThan(
	valueToTest := THIS^.DATE_LSB_IS_UNSET,
	lessValue := THIS^.DATE_MAX
);
THIS^.testValueIsGreaterThan(
	valueToTest := THIS^.DATE_MAX,
	lessValue := THIS^.DATE_LSB_IS_UNSET
);
TcUnit.TEST_FINISHED();
END_METHOD

(*

short summary
==================
This test method tests ``assert.dateAndTime.simple.dateOnly.valueIsInRangeOf``
method of CNM_AssertionInterfaceLib library with various inputs

.. <legal notes>

legal notes
=================
| SPDX-FileCopyrightText: © 2022 ekvip automation GmbH <info@ekvip.de>
| SPDX-License-Identifier: Apache-2.0
| For details check: Apache-2.0_

.. _Apache-2.0: https://www.apache.org/licenses/LICENSE-2.0

.. </legal notes>

*)

METHOD runValueIsInRangeOfTests
RETURN (NOT TcUnit.TEST_ORDERED(THIS^.getTestNameFor('valueIsInRangeOf')));

THIS^.testValueIsInRangeOf(
	lowerLimit := THIS^.DATE_MIN,
	valueToTest := THIS^.DATE_MAX,
	upperLimit	:= THIS^.DATE_MAX
);
THIS^.testValueIsInRangeOf(
	lowerLimit := THIS^.DATE_MIN,
	valueToTest := THIS^.DATE_MIN,
	upperLimit	:= THIS^.DATE_MAX
);
THIS^.testValueIsInRangeOf(
	lowerLimit := THIS^.DATE_MAX,
	valueToTest := THIS^.DATE_MAX,
	upperLimit	:= THIS^.DATE_MIN
);
THIS^.testValueIsInRangeOf(
	lowerLimit := THIS^.DATE_MAX,
	valueToTest := THIS^.DATE_MIN,
	upperLimit	:= THIS^.DATE_MIN
);
THIS^.testValueIsInRangeOf(
	lowerLimit := THIS^.DATE_LSB_IS_UNSET,
	valueToTest := THIS^.DATE_MIN,
	upperLimit	:= THIS^.DATE_MAX
);
THIS^.testValueIsInRangeOf(
	lowerLimit := THIS^.DATE_MIN,
	valueToTest := THIS^.DATE_LSB_IS_UNSET,
	upperLimit	:= THIS^.DATE_MAX
);
THIS^.testValueIsInRangeOf(
	lowerLimit := THIS^.DATE_LSB_IS_UNSET,
	valueToTest := THIS^.DATE_LSB_IS_UNSET,
	upperLimit	:= THIS^.DATE_LSB_IS_UNSET
);
THIS^.testValueIsInRangeOf(
	lowerLimit := THIS^.DATE_ALL_NIBBLE_LSB,
	valueToTest := THIS^.DATE_LSB_IS_UNSET,
	upperLimit	:= THIS^.DATE_ALL_NIBBLE_MSB
);
THIS^.testValueIsInRangeOf(
	lowerLimit := THIS^.DATE_LSB_IS_UNSET,
	valueToTest := THIS^.DATE_ALL_NIBBLE_LSB,
	upperLimit	:= THIS^.DATE_ALL_NIBBLE_MSB
);
THIS^.testValueIsInRangeOf(
	lowerLimit := THIS^.DATE_LSB_ONLY,
	valueToTest := THIS^.DATE_WITHOUT_MSB,
	upperLimit	:= THIS^.DATE_MSB_ONLY
);
THIS^.testValueIsInRangeOf(
	lowerLimit := THIS^.DATE_WITHOUT_MSB,
	valueToTest := THIS^.DATE_LSB_ONLY,
	upperLimit	:= THIS^.DATE_MSB_ONLY
);
THIS^.testValueIsInRangeOf(
	lowerLimit := THIS^.DATE_WITHOUT_NIBBLE_MSB,
	valueToTest := THIS^.DATE_MAX,
	upperLimit	:= THIS^.DATE_ALL_NIBBLE_MSB
);
THIS^.testValueIsInRangeOf(
	lowerLimit := THIS^.DATE_WITHOUT_NIBBLE_MSB,
	valueToTest := THIS^.DATE_MIN,
	upperLimit	:= THIS^.DATE_ALL_NIBBLE_MSB
);
THIS^.testValueIsInRangeOf(
	lowerLimit := THIS^.DATE_WITHOUT_NIBBLE_MSB,
	valueToTest := THIS^.DATE_WITHOUT_NIBBLE_MSB,
	upperLimit	:= THIS^.DATE_ALL_NIBBLE_MSB
);
THIS^.testValueIsInRangeOf(
	lowerLimit := THIS^.DATE_WITHOUT_NIBBLE_MSB,
	valueToTest := THIS^.DATE_ALL_NIBBLE_MSB,
	upperLimit	:= THIS^.DATE_ALL_NIBBLE_MSB
);
TcUnit.TEST_FINISHED();
END_METHOD

(*

short summary
==================
This test method tests ``assert.dateAndTime.simple.dateOnly.valueIsLessThan``
method of CNM_AssertionInterfaceLib library with various inputs

.. <legal notes>

legal notes
=================
| SPDX-FileCopyrightText: © 2022 ekvip automation GmbH <info@ekvip.de>
| SPDX-License-Identifier: Apache-2.0
| For details check: Apache-2.0_

.. _Apache-2.0: https://www.apache.org/licenses/LICENSE-2.0

.. </legal notes>

*)

METHOD runValueIsLessThanTests
RETURN (NOT TcUnit.TEST_ORDERED(THIS^.getTestNameFor('valueIsLessThan')));

THIS^.testValueIsLessThan(
	valueToTest := THIS^.DATE_MAX,
	greaterValue := THIS^.DATE_MAX
);
THIS^.testValueIsLessThan(
	valueToTest := THIS^.DATE_MIN,
	greaterValue := THIS^.DATE_MIN
);
THIS^.testValueIsLessThan(
	valueToTest := THIS^.DATE_MIN,
	greaterValue := THIS^.DATE_MAX
);
THIS^.testValueIsLessThan(
	valueToTest := THIS^.DATE_MAX,
	greaterValue := THIS^.DATE_MIN
);
THIS^.testValueIsLessThan(
	valueToTest := THIS^.DATE_ALL_NIBBLE_LSB,
	greaterValue := THIS^.DATE_ALL_NIBBLE_LSB
);
THIS^.testValueIsLessThan(
	valueToTest := THIS^.DATE_ALL_NIBBLE_MSB,
	greaterValue := THIS^.DATE_ALL_NIBBLE_LSB
);
THIS^.testValueIsLessThan(
	valueToTest := THIS^.DATE_ALL_NIBBLE_LSB,
	greaterValue := THIS^.DATE_ALL_NIBBLE_MSB
);
THIS^.testValueIsLessThan(
	valueToTest := THIS^.DATE_LSB_ONLY,
	greaterValue := THIS^.DATE_MSB_ONLY
);
THIS^.testValueIsLessThan(
	valueToTest := THIS^.DATE_MSB_ONLY,
	greaterValue := THIS^.DATE_MSB_ONLY
);
THIS^.testValueIsLessThan(
	valueToTest := THIS^.DATE_MSB_ONLY,
	greaterValue := THIS^.DATE_LSB_ONLY
);
THIS^.testValueIsLessThan(
	valueToTest := THIS^.DATE_LSB_IS_UNSET,
	greaterValue := THIS^.DATE_MAX
);
THIS^.testValueIsLessThan(
	valueToTest := THIS^.DATE_MAX,
	greaterValue := THIS^.DATE_LSB_IS_UNSET
);
TcUnit.TEST_FINISHED();
END_METHOD

(*

short summary
==================
This test method tests ``assert.dateAndTime.simple.dateOnly.valueIsMax``
method of CNM_AssertionInterfaceLib library with various inputs

.. <legal notes>

legal notes
=================
| SPDX-FileCopyrightText: © 2022 ekvip automation GmbH <info@ekvip.de>
| SPDX-License-Identifier: Apache-2.0
| For details check: Apache-2.0_

.. _Apache-2.0: https://www.apache.org/licenses/LICENSE-2.0

.. </legal notes>

*)

METHOD runValueIsMaxTests
RETURN (NOT TcUnit.TEST_ORDERED(THIS^.getTestNameFor('valueIsMax')));

THIS^.testValueIsMax(
	valueToTest := THIS^.DATE_MAX,
	maximumValue := THIS^.DATE_MAX
);
THIS^.testValueIsMax(
	valueToTest := THIS^.DATE_MIN,
	maximumValue := THIS^.DATE_MIN
);
THIS^.testValueIsMax(
	valueToTest := THIS^.DATE_MIN,
	maximumValue := THIS^.DATE_MAX
);
THIS^.testValueIsMax(
	valueToTest := THIS^.DATE_MAX,
	maximumValue := THIS^.DATE_MIN
);
THIS^.testValueIsMax(
	valueToTest := THIS^.DATE_ALL_NIBBLE_LSB,
	maximumValue := THIS^.DATE_ALL_NIBBLE_LSB
);
THIS^.testValueIsMax(
	valueToTest := THIS^.DATE_ALL_NIBBLE_MSB,
	maximumValue := THIS^.DATE_ALL_NIBBLE_LSB
);
THIS^.testValueIsMax(
	valueToTest := THIS^.DATE_ALL_NIBBLE_LSB,
	maximumValue := THIS^.DATE_ALL_NIBBLE_MSB
);
THIS^.testValueIsMax(
	valueToTest := THIS^.DATE_LSB_ONLY,
	maximumValue := THIS^.DATE_MSB_ONLY
);
THIS^.testValueIsMax(
	valueToTest := THIS^.DATE_MSB_ONLY,
	maximumValue := THIS^.DATE_MSB_ONLY
);
THIS^.testValueIsMax(
	valueToTest := THIS^.DATE_MSB_ONLY,
	maximumValue := THIS^.DATE_LSB_ONLY
);
THIS^.testValueIsMax(
	valueToTest := THIS^.DATE_LSB_IS_UNSET,
	maximumValue := THIS^.DATE_MAX
);
THIS^.testValueIsMax(
	valueToTest := THIS^.DATE_MAX,
	maximumValue := THIS^.DATE_LSB_IS_UNSET
);
TcUnit.TEST_FINISHED();
END_METHOD

(*

short summary
==================
This test method tests ``assert.dateAndTime.simple.dateOnly.valueIsMin``
method of CNM_AssertionInterfaceLib library with various inputs

.. <legal notes>

legal notes
=================
| SPDX-FileCopyrightText: © 2022 ekvip automation GmbH <info@ekvip.de>
| SPDX-License-Identifier: Apache-2.0
| For details check: Apache-2.0_

.. _Apache-2.0: https://www.apache.org/licenses/LICENSE-2.0

.. </legal notes>

*)

METHOD runValueIsMinTests
RETURN (NOT TcUnit.TEST_ORDERED(THIS^.getTestNameFor('valueIsMin')));

THIS^.testValueIsMin(
	valueToTest := THIS^.DATE_MAX,
	minimumValue := THIS^.DATE_MAX
);
THIS^.testValueIsMin(
	valueToTest := THIS^.DATE_MIN,
	minimumValue := THIS^.DATE_MIN
);
THIS^.testValueIsMin(
	valueToTest := THIS^.DATE_MIN,
	minimumValue := THIS^.DATE_MAX
);
THIS^.testValueIsMin(
	valueToTest := THIS^.DATE_MAX,
	minimumValue := THIS^.DATE_MIN
);
THIS^.testValueIsMin(
	valueToTest := THIS^.DATE_ALL_NIBBLE_LSB,
	minimumValue := THIS^.DATE_ALL_NIBBLE_LSB
);
THIS^.testValueIsMin(
	valueToTest := THIS^.DATE_ALL_NIBBLE_MSB,
	minimumValue := THIS^.DATE_ALL_NIBBLE_LSB
);
THIS^.testValueIsMin(
	valueToTest := THIS^.DATE_ALL_NIBBLE_LSB,
	minimumValue := THIS^.DATE_ALL_NIBBLE_MSB
);
THIS^.testValueIsMin(
	valueToTest := THIS^.DATE_LSB_ONLY,
	minimumValue := THIS^.DATE_MSB_ONLY
);
THIS^.testValueIsMin(
	valueToTest := THIS^.DATE_MSB_ONLY,
	minimumValue := THIS^.DATE_MSB_ONLY
);
THIS^.testValueIsMin(
	valueToTest := THIS^.DATE_MSB_ONLY,
	minimumValue := THIS^.DATE_LSB_ONLY
);
THIS^.testValueIsMin(
	valueToTest := THIS^.DATE_LSB_IS_UNSET,
	minimumValue := THIS^.DATE_MAX
);
THIS^.testValueIsMin(
	valueToTest := THIS^.DATE_MAX,
	minimumValue := THIS^.DATE_LSB_IS_UNSET
);
TcUnit.TEST_FINISHED();
END_METHOD

(*

short summary
==================
This test method tests ``assert.dateAndTime.simple.dateOnly.valueIsNotEqualTo``
method of CNM_AssertionInterfaceLib library with various inputs

.. <legal notes>

legal notes
=================
| SPDX-FileCopyrightText: © 2022 ekvip automation GmbH <info@ekvip.de>
| SPDX-License-Identifier: Apache-2.0
| For details check: Apache-2.0_

.. _Apache-2.0: https://www.apache.org/licenses/LICENSE-2.0

.. </legal notes>

*)

METHOD runValueIsNotEqualToTests
RETURN (NOT TcUnit.TEST_ORDERED(THIS^.getTestNameFor('valueIsNotEqualTo')));

THIS^.testValueIsNotEqualTo(
	valueToTest := THIS^.DATE_MAX,
	unexpectedValue := THIS^.DATE_MAX
);
THIS^.testValueIsNotEqualTo(
	valueToTest := THIS^.DATE_MIN,
	unexpectedValue := THIS^.DATE_MIN
);
THIS^.testValueIsNotEqualTo(
	valueToTest := THIS^.DATE_MIN,
	unexpectedValue := THIS^.DATE_MAX
);
THIS^.testValueIsNotEqualTo(
	valueToTest := THIS^.DATE_MAX,
	unexpectedValue := THIS^.DATE_MIN
);
THIS^.testValueIsNotEqualTo(
	valueToTest := THIS^.DATE_ALL_NIBBLE_LSB,
	unexpectedValue := THIS^.DATE_ALL_NIBBLE_LSB
);
THIS^.testValueIsNotEqualTo(
	valueToTest := THIS^.DATE_LSB_ONLY,
	unexpectedValue := THIS^.DATE_MSB_ONLY
);
THIS^.testValueIsNotEqualTo(
	valueToTest := THIS^.DATE_MSB_ONLY,
	unexpectedValue := THIS^.DATE_MSB_ONLY
);
THIS^.testValueIsNotEqualTo(
	valueToTest := THIS^.DATE_MSB_ONLY,
	unexpectedValue := THIS^.DATE_LSB_ONLY
);

TcUnit.TEST_FINISHED();
END_METHOD

(*

short summary
==================
This test method tests ``assert.dateAndTime.simple.dateOnly.valueIsEqualTo``
method of CNM_AssertionInterfaceLib library, 
it provides the possibility to handover test data via parameter 


.. <legal notes>

legal notes
=================
| SPDX-FileCopyrightText: © 2022 ekvip automation GmbH <info@ekvip.de>
| SPDX-License-Identifier: Apache-2.0
| For details check: Apache-2.0_

.. _Apache-2.0: https://www.apache.org/licenses/LICENSE-2.0

.. </legal notes>

parameters
==========

*)

METHOD testValueIsEqualTo 
VAR_INPUT
	(* for the test it's the parameter ``currentValue`` *)
	valueToTest	:DATE;
	(* for the test it's the parameter ``expectedValue`` *)
	expected	:DATE;
END_VAR
VAR
	(* just the expectation if the assertion to test must be worng or true *)
	assertionIsWrong		:BOOL;
	(* contains the format string for the test message *)
	message					:Tc2_System.T_MaxString;
	(* TwinCAT printf with the test message *)
	messageStringBuilder	:Tc2_Utilities.FB_FormatString;
	(* DATE value of ``currentValue`` as string *)
	currentValueAsString	:STRING(22);
	(* DATE value of ``expectedValue`` as string *)
	expectedValueAsString	:STRING(22);
END_VAR
THIS^.assertorContainer.resetAssertor();

assertionIsWrong := (valueToTest <> expected);
message := SEL(
	assertionIsWrong,
	'currentValue is %s expectedValue is %s assertion must be TRUE', 
	'currentValue is %s expectedValue is %s assertion must be FALSE'
);
currentValueAsString := TO_STRING(valueToTest);
expectedValueAsString := TO_STRING(expected);

messageStringBuilder(
	sFormat := message,
	arg1 := THIS^.AnyToArg(currentValueAsString),
	arg2 := THIS^.AnyToArg(expectedValueAsString)
);

THIS^.assertorContainer.assertor.assert.dateAndTime.simple.dateOnly.valueIsEqualTo(
	currentValue	:= valueToTest,
	expectedValue	:= expected,
	message			:= ''
   );

THIS^.AssertEquals_BOOL(
	Expected 	:= assertionIsWrong,
	Actual 		:= THIS^.assertorContainer.wasAssertionWrong,
	Message 	:= messageStringBuilder.sOut
);
END_METHOD

(*

short summary
==================
This test method tests ``assert.dateAndTime.simple.dateOnly.valueIsGreaterThan``
method of CNM_AssertionInterfaceLib library, 
it provides the possibility to handover test data via parameter 


.. <legal notes>

legal notes
=================
| SPDX-FileCopyrightText: © 2022 ekvip automation GmbH <info@ekvip.de>
| SPDX-License-Identifier: Apache-2.0
| For details check: Apache-2.0_

.. _Apache-2.0: https://www.apache.org/licenses/LICENSE-2.0

.. </legal notes>

parameters
==========

*)

METHOD testValueIsGreaterThan 
VAR_INPUT
	(* for the test it's the parameter ``currentValue`` *)
	valueToTest	:DATE;
	(* for the test it's the parameter ``lessValue`` *)
	lessValue	:DATE;
END_VAR
VAR
	(* just the expectation if the assertion to test must be worng or true *)
	assertionIsWrong		:BOOL;
	(* contains the format string for the test message *)
	message					:Tc2_System.T_MaxString;
	(* TwinCAT printf with the test message *)
	messageStringBuilder	:Tc2_Utilities.FB_FormatString;
	(* DATE value of ``currentValue`` as string *)
	currentValueAsString	:STRING(22);
	(* DATE value of ``lessValue`` as string *)
	lessValueAsString		:STRING(22);
END_VAR
THIS^.assertorContainer.resetAssertor();

assertionIsWrong := (valueToTest <= lessValue);
message := SEL(
	assertionIsWrong,
	'currentValue is %s lessValue is %s assertion must be TRUE', 
	'currentValue is %s lessValue is %s assertion must be FALSE'
);
currentValueAsString := TO_STRING(valueToTest);
lessValueAsString := TO_STRING(lessValue);

messageStringBuilder(
	sFormat := message,
	arg1 := THIS^.AnyToArg(currentValueAsString),
	arg2 := THIS^.AnyToArg(lessValueAsString)
);

THIS^.assertorContainer.assertor.assert.dateAndTime.simple.dateOnly.valueIsGreaterThan(
	currentValue	:= valueToTest,
	lessValue		:= lessValue,
	message			:= ''
   );

THIS^.AssertEquals_BOOL(
	Expected 	:= assertionIsWrong,
	Actual 		:= THIS^.assertorContainer.wasAssertionWrong,
	Message 	:= messageStringBuilder.sOut
);
END_METHOD

(*

short summary
==================
This test method tests ``assert.dateAndTime.simple.dateOnly.valueIsInRangeOf``
method of CNM_AssertionInterfaceLib library, 
it provides the possibility to handover test data via parameter 


.. <legal notes>

legal notes
=================
| SPDX-FileCopyrightText: © 2022 ekvip automation GmbH <info@ekvip.de>
| SPDX-License-Identifier: Apache-2.0
| For details check: Apache-2.0_

.. _Apache-2.0: https://www.apache.org/licenses/LICENSE-2.0

.. </legal notes>

parameters
==========

*)

METHOD testValueIsInRangeOf 
VAR_INPUT
	(* for the test it's the parameter ``lowerLimit`` *)
	lowerLimit	:DATE;
	(* for the test it's the parameter ``currentValue`` *)
	valueToTest	:DATE;
	(* for the test it's the parameter ``upperLimit`` *)
	upperLimit	:DATE;
END_VAR
VAR
	(* just the expectation if the assertion to test must be worng or true *)
	assertionIsWrong		:BOOL;
	(* contains the format string for the test message *)
	message					:Tc2_System.T_MaxString;
	(* TwinCAT printf with the test message *)
	messageStringBuilder	:Tc2_Utilities.FB_FormatString;
	(* DATE value of ``lowerLimit`` as string *)
	lowerLimitAsString		:STRING(22);
	(* DATE value of ``currentValue`` as string *)
	currentValueAsString	:STRING(22);
	(* DATE value of ``upperLimit`` as string *)
	upperLimitAsString		:STRING(22);

END_VAR
THIS^.assertorContainer.resetAssertor();

assertionIsWrong := ((valueToTest < lowerLimit) OR (valueToTest > upperLimit));
message := SEL(
	assertionIsWrong,
	'lowerLimit is %s currentValue is %s upperLimit is %s assertion must be TRUE', 
	'lowerLimit is %s currentValue is %s upperLimit is %s assertion must be FALSE'
);
lowerLimitAsString		:= TO_STRING(lowerLimit);
currentValueAsString	:= TO_STRING(valueToTest);
upperLimitAsString		:= TO_STRING(upperLimit);

messageStringBuilder(
	sFormat := message,
	arg1 := THIS^.AnyToArg(lowerLimitAsString),
	arg2 := THIS^.AnyToArg(currentValueAsString),
	arg3 := THIS^.AnyToArg(upperLimitAsString)
);

THIS^.assertorContainer.assertor.assert.dateAndTime.simple.dateOnly.valueIsInRangeOf(
	lowerLimit		:= lowerLimit,
	currentValue	:= valueToTest,
	upperLimit		:= upperLimit,
	message			:= ''
   );

THIS^.AssertEquals_BOOL(
	Expected 	:= assertionIsWrong,
	Actual 		:= THIS^.assertorContainer.wasAssertionWrong,
	Message 	:= messageStringBuilder.sOut
);
END_METHOD

(*

short summary
==================
This test method tests ``assert.dateAndTime.simple.dateOnly.valueIsLessThan``
method of CNM_AssertionInterfaceLib library, 
it provides the possibility to handover test data via parameter 


.. <legal notes>

legal notes
=================
| SPDX-FileCopyrightText: © 2022 ekvip automation GmbH <info@ekvip.de>
| SPDX-License-Identifier: Apache-2.0
| For details check: Apache-2.0_

.. _Apache-2.0: https://www.apache.org/licenses/LICENSE-2.0

.. </legal notes>

parameters
==========

*)

METHOD testValueIsLessThan 
VAR_INPUT
	(* for the test it's the parameter ``currentValue`` *)
	valueToTest		:DATE;
	(* for the test it's the parameter ``greaterValue`` *)
	greaterValue	:DATE;
END_VAR
VAR
	(* just the expectation if the assertion to test must be worng or true *)
	assertionIsWrong		:BOOL;
	(* contains the format string for the test message *)
	message					:Tc2_System.T_MaxString;
	(* TwinCAT printf with the test message *)
	messageStringBuilder	:Tc2_Utilities.FB_FormatString;
	(* DATE value of ``currentValue`` as string *)
	currentValueAsString	:STRING(22);
	(* DATE value of ``greaterValue`` as string *)
	greaterValueAsString	:STRING(22);
END_VAR
THIS^.assertorContainer.resetAssertor();

assertionIsWrong := (valueToTest >= greaterValue);
message := SEL(
	assertionIsWrong,
	'currentValue is %s greaterValue is %s assertion must be TRUE', 
	'currentValue is %s greaterValue is %s assertion must be FALSE'
);
currentValueAsString := TO_STRING(valueToTest);
greaterValueAsString := TO_STRING(greaterValue);

messageStringBuilder(
	sFormat := message,
	arg1 := THIS^.AnyToArg(currentValueAsString),
	arg2 := THIS^.AnyToArg(greaterValueAsString)
);

THIS^.assertorContainer.assertor.assert.dateAndTime.simple.dateOnly.valueIsLessThan(
	currentValue	:= valueToTest,
	greaterValue	:= greaterValue,
	message			:= ''
   );

THIS^.AssertEquals_BOOL(
	Expected 	:= assertionIsWrong,
	Actual 		:= THIS^.assertorContainer.wasAssertionWrong,
	Message 	:= messageStringBuilder.sOut
);
END_METHOD

(*

short summary
==================
This test method tests ``assert.dateAndTime.simple.dateOnly.valueIsMax``
method of CNM_AssertionInterfaceLib library, 
it provides the possibility to handover test data via parameter 


.. <legal notes>

legal notes
=================
| SPDX-FileCopyrightText: © 2022 ekvip automation GmbH <info@ekvip.de>
| SPDX-License-Identifier: Apache-2.0
| For details check: Apache-2.0_

.. _Apache-2.0: https://www.apache.org/licenses/LICENSE-2.0

.. </legal notes>

parameters
==========

*)

METHOD testValueIsMax 
VAR_INPUT
	(* for the test it's the parameter ``currentValue`` *)
	valueToTest		:DATE;
	(* for the test it's the parameter ``greaterValue`` *)
	maximumValue	:DATE;
END_VAR
VAR
	(* just the expectation if the assertion to test must be worng or true *)
	assertionIsWrong		:BOOL;
	(* contains the format string for the test message *)
	message					:Tc2_System.T_MaxString;
	(* TwinCAT printf with the test message *)
	messageStringBuilder	:Tc2_Utilities.FB_FormatString;
	(* DATE value of ``currentValue`` as string *)
	currentValueAsString	:STRING(22);
	(* DATE value of ``maximumValue`` as string *)
	maximumValueAsString	:STRING(22);
END_VAR
THIS^.assertorContainer.resetAssertor();

assertionIsWrong := (valueToTest > maximumValue);
message := SEL(
	assertionIsWrong,
	'currentValue is %s maximumValue is %s assertion must be TRUE', 
	'currentValue is %s maximumValue is %s assertion must be FALSE'
);
currentValueAsString := TO_STRING(valueToTest);
maximumValueAsString := TO_STRING(maximumValue);

messageStringBuilder(
	sFormat := message,
	arg1 := THIS^.AnyToArg(currentValueAsString),
	arg2 := THIS^.AnyToArg(maximumValueAsString)
);

THIS^.assertorContainer.assertor.assert.dateAndTime.simple.dateOnly.valueIsMax(
	currentValue	:= valueToTest,
	maximumValue	:= maximumValue,
	message			:= ''
   );

THIS^.AssertEquals_BOOL(
	Expected 	:= assertionIsWrong,
	Actual 		:= THIS^.assertorContainer.wasAssertionWrong,
	Message 	:= messageStringBuilder.sOut
);
END_METHOD

(*

short summary
==================
This test method tests ``assert.dateAndTime.simple.dateOnly.valueIsMin``
method of CNM_AssertionInterfaceLib library, 
it provides the possibility to handover test data via parameter 


.. <legal notes>

legal notes
=================
| SPDX-FileCopyrightText: © 2022 ekvip automation GmbH <info@ekvip.de>
| SPDX-License-Identifier: Apache-2.0
| For details check: Apache-2.0_

.. _Apache-2.0: https://www.apache.org/licenses/LICENSE-2.0

.. </legal notes>

parameters
==========

*)

METHOD testValueIsMin 
VAR_INPUT
	(* for the test it's the parameter ``currentValue`` *)
	valueToTest		:DATE;
	(* for the test it's the parameter ``greaterValue`` *)
	minimumValue	:DATE;
END_VAR
VAR
	(* just the expectation if the assertion to test must be worng or true *)
	assertionIsWrong		:BOOL;
	(* contains the format string for the test message *)
	message					:Tc2_System.T_MaxString;
	(* TwinCAT printf with the test message *)
	messageStringBuilder	:Tc2_Utilities.FB_FormatString;
	(* DATE value of ``currentValue`` as string *)
	currentValueAsString	:STRING(22);
	(* DATE value of ``minimumValue`` as string *)
	minimumValueAsString	:STRING(22);
END_VAR
THIS^.assertorContainer.resetAssertor();

assertionIsWrong := (valueToTest < minimumValue);
message := SEL(
	assertionIsWrong,
	'currentValue is %s minimumValue is %s assertion must be TRUE', 
	'currentValue is %s minimumValue is %s assertion must be FALSE'
);
currentValueAsString := TO_STRING(valueToTest);
minimumValueAsString := TO_STRING(minimumValue);

messageStringBuilder(
	sFormat := message,
	arg1 := THIS^.AnyToArg(currentValueAsString),
	arg2 := THIS^.AnyToArg(minimumValueAsString)
);

THIS^.assertorContainer.assertor.assert.dateAndTime.simple.dateOnly.valueIsMin(
	currentValue	:= valueToTest,
	minimumValue	:= minimumValue,
	message			:= ''
   );

THIS^.AssertEquals_BOOL(
	Expected 	:= assertionIsWrong,
	Actual 		:= THIS^.assertorContainer.wasAssertionWrong,
	Message 	:= messageStringBuilder.sOut
);
END_METHOD

(*

short summary
==================
This test method tests ``assert.dateAndTime.simple.dateOnly.valueIsNotEqualTo``
method of CNM_AssertionInterfaceLib library, 
it provides the possibility to handover test data via parameter 


.. <legal notes>

legal notes
=================
| SPDX-FileCopyrightText: © 2022 ekvip automation GmbH <info@ekvip.de>
| SPDX-License-Identifier: Apache-2.0
| For details check: Apache-2.0_

.. _Apache-2.0: https://www.apache.org/licenses/LICENSE-2.0

.. </legal notes>

parameters
==========

*)

METHOD testValueIsNotEqualTo 
VAR_INPUT
	(* for the test it's the parameter ``currentValue`` *)
	valueToTest		:DATE;
	(* for the test it's the parameter ``unexpectedValue`` *)
	unexpectedValue	:DATE;
END_VAR
VAR
	(* just the expectation if the assertion to test must be worng or true *)
	assertionIsWrong		:BOOL;
	(* contains the format string for the test message *)
	message					:Tc2_System.T_MaxString;
	(* TwinCAT printf with the test message *)
	messageStringBuilder	:Tc2_Utilities.FB_FormatString;
	(* DATE value of ``currentValue`` as string *)
	currentValueAsString	:STRING(22);
	(* DATE value of ``unexpectedValue`` as string *)
	unexpectedValueAsString	:STRING(22);
END_VAR
THIS^.assertorContainer.resetAssertor();

assertionIsWrong := (valueToTest = unexpectedValue);
message := SEL(
	assertionIsWrong,
	'currentValue is %s expectedValue is %s assertion must be TRUE', 
	'currentValue is %s expectedValue is %s assertion must be FALSE'
);
currentValueAsString := TO_STRING(valueToTest);
unexpectedValueAsString := TO_STRING(unexpectedValue);

messageStringBuilder(
	sFormat := message,
	arg1 := THIS^.AnyToArg(currentValueAsString),
	arg2 := THIS^.AnyToArg(unexpectedValueAsString)
);

THIS^.assertorContainer.assertor.assert.dateAndTime.simple.dateOnly.valueIsNotEqualTo(
	currentValue	:= valueToTest,
	unexpectedValue	:= unexpectedValue,
	message			:= ''
   );

THIS^.AssertEquals_BOOL(
	Expected 	:= assertionIsWrong,
	Actual 		:= THIS^.assertorContainer.wasAssertionWrong,
	Message 	:= messageStringBuilder.sOut
);
END_METHOD

END_FUNCTION_BLOCK

// ---- AssertionTester/AssertionTests/DateTimeAssertions/classes/TODAssertionTests.TcPOU
(*

short summary
==================
This class tests all methods of TOD assertions
with various combinations of inputs and checks expected 
outputs are satisfied or not

.. <legal notes>

legal notes
=================
| SPDX-FileCopyrightText: © 2022 ekvip automation GmbH <info@ekvip.de>
| SPDX-License-Identifier: Apache-2.0
| For details check: Apache-2.0_

.. _Apache-2.0: https://www.apache.org/licenses/LICENSE-2.0

.. </legal notes>

methods and properties
======================

*)


FUNCTION_BLOCK TODAssertionTests EXTENDS AbstractAssertorTest
VAR
	
END_VAR
VAR CONSTANT
	(* prefix to unify the test names *)
	TEST_NAME_PREFIX		:STRING := 'assert.dateAndTime.simple.timeOfDay.';
	(* max value of a DWORD *)
	{attribute 'hide'}
	MAX_DWORD				:DWORD := 16#FFFF_FFFF;
	(* min value of a DWORD *)
	{attribute 'hide'}
	MIN_DWORD				:DWORD := 16#0000_0000;
	(* only the msb is set *)
	{attribute 'hide'}
	MSB_ONLY				:DWORD := 16#8000_0000;
	(* only the msb is set *)
	{attribute 'hide'}
	LSB_ONLY				:DWORD := 16#0000_0001;
	(* all bits set except the msb *)
	{attribute 'hide'}
	WITHOUT_MSB 			:DWORD := 16#7FFF_FFFF;
	(* for every nibble is the msb set only *)
	{attribute 'hide'}
	ALL_NIBBLE_MSB			:DWORD := 16#8888_8888;
	(* for every nibble is the msb unset only *)
	{attribute 'hide'}
	WITHOUT_NIBBLE_MSB		:DWORD := 16#7777_7777;
	(* for every nibble is the lsb set only *)
	{attribute 'hide'}
	ALL_NIBBLE_LSB			:DWORD := 16#1111_1111;
	(* every bit is set except the lsb *)
	{attribute 'hide'}
	LSB_IS_UNSET			:DWORD := 16#FFFF_FFFE;
	(* max vale of time of day *)
	TOD_MAX					:TOD := TO_TOD(MAX_DWORD);
	(* min vale of time of day *)
	TOD_MIN					:TOD := TO_TOD(MIN_DWORD);
	(* only the msb is set *)
	TOD_MSB_ONLY			:TOD := TO_TOD(MSB_ONLY);
	(* all bits set except the msb *)
	TOD_WITHOUT_MSB 		:TOD := TO_TOD(WITHOUT_MSB);
	(* for every nibble is the msb set only *)
	TOD_ALL_NIBBLE_MSB		:TOD := TO_TOD(ALL_NIBBLE_MSB);
	(* for every nibble is the msb unset only *)
	TOD_WITHOUT_NIBBLE_MSB	:TOD := TO_TOD(WITHOUT_NIBBLE_MSB);
	(* for every nibble is the lsb set only *)
	TOD_ALL_NIBBLE_LSB		:TOD := TO_TOD(ALL_NIBBLE_LSB);	
	(* every bit is set except the lsb *)
	TOD_LSB_IS_UNSET		:TOD := TO_TOD(LSB_IS_UNSET);
	(* only the msb is set *)
	TOD_LSB_ONLY			:TOD := TO_TOD(LSB_ONLY);
END_VAR

THIS^.runValueIsEqualToTests();
THIS^.runValueIsGreaterThanTests();
THIS^.runValueIsInRangeOfTests();
THIS^.runValueIsLessThanTests();
THIS^.runValueIsMaxTests();
THIS^.runValueIsMinTests();
THIS^.runValueIsNotEqualToTests();

(*

short summary
==================
This test method is a helper function to create a unified test name

.. <legal notes>

legal notes
=================
| SPDX-FileCopyrightText: © 2022 ekvip automation GmbH <info@ekvip.de>
| SPDX-License-Identifier: Apache-2.0
| For details check: Apache-2.0_

.. _Apache-2.0: https://www.apache.org/licenses/LICENSE-2.0

.. </legal notes>

parameters
==========

*)

METHOD PROTECTED getTestNameFor :Tc2_System.T_MaxString
VAR_INPUT
	(* name of the method to test, to create a unified test name *)
	nameOfMethodToTest	:Tc2_System.T_MaxString;
END_VAR
getTestNameFor := Tc2_Standard.CONCAT(THIS^.TEST_NAME_PREFIX, nameOfMethodToTest);
END_METHOD

(*

short summary
==================
This test method tests ``assert.dateAndTime.simple.timeOfDay.valueIsEqualTo``
method of CNM_AssertionInterfaceLib library with various inputs

.. <legal notes>

legal notes
=================
| SPDX-FileCopyrightText: © 2022 ekvip automation GmbH <info@ekvip.de>
| SPDX-License-Identifier: Apache-2.0
| For details check: Apache-2.0_

.. _Apache-2.0: https://www.apache.org/licenses/LICENSE-2.0

.. </legal notes>

*)

METHOD runValueIsEqualToTests
RETURN (NOT TcUnit.TEST_ORDERED(THIS^.getTestNameFor('valueIsEqualTo')));

THIS^.testValueIsEqualTo(
	valueToTest := THIS^.TOD_MAX,
	expected := THIS^.TOD_MAX
);
THIS^.testValueIsEqualTo(
	valueToTest := THIS^.TOD_MIN,
	expected := THIS^.TOD_MIN
);
THIS^.testValueIsEqualTo(
	valueToTest := THIS^.TOD_MIN,
	expected := THIS^.TOD_MAX
);
THIS^.testValueIsEqualTo(
	valueToTest := THIS^.TOD_MAX,
	expected := THIS^.TOD_MIN
);
THIS^.testValueIsEqualTo(
	valueToTest := THIS^.TOD_ALL_NIBBLE_LSB,
	expected := THIS^.TOD_ALL_NIBBLE_LSB
);
THIS^.testValueIsEqualTo(
	valueToTest := THIS^.TOD_LSB_ONLY,
	expected := THIS^.TOD_MSB_ONLY
);
THIS^.testValueIsEqualTo(
	valueToTest := THIS^.TOD_MSB_ONLY,
	expected := THIS^.TOD_MSB_ONLY
);
THIS^.testValueIsEqualTo(
	valueToTest := THIS^.TOD_MSB_ONLY,
	expected := THIS^.TOD_LSB_ONLY
);

TcUnit.TEST_FINISHED();
END_METHOD

(*

short summary
==================
This test method tests ``assert.dateAndTime.simple.timeOfDay.valueIsGreaterThan``
method of CNM_AssertionInterfaceLib library with various inputs

.. <legal notes>

legal notes
=================
| SPDX-FileCopyrightText: © 2022 ekvip automation GmbH <info@ekvip.de>
| SPDX-License-Identifier: Apache-2.0
| For details check: Apache-2.0_

.. _Apache-2.0: https://www.apache.org/licenses/LICENSE-2.0

.. </legal notes>

*)

METHOD runValueIsGreaterThanTests
RETURN (NOT TcUnit.TEST_ORDERED(THIS^.getTestNameFor('valueIsGreaterThan')));

THIS^.testValueIsGreaterThan(
	valueToTest := THIS^.TOD_MAX,
	lessValue := THIS^.TOD_MAX
);
THIS^.testValueIsGreaterThan(
	valueToTest := THIS^.TOD_MIN,
	lessValue := THIS^.TOD_MIN
);
THIS^.testValueIsGreaterThan(
	valueToTest := THIS^.TOD_MIN,
	lessValue := THIS^.TOD_MAX
);
THIS^.testValueIsGreaterThan(
	valueToTest := THIS^.TOD_MAX,
	lessValue := THIS^.TOD_MIN
);
THIS^.testValueIsGreaterThan(
	valueToTest := THIS^.TOD_ALL_NIBBLE_LSB,
	lessValue := THIS^.TOD_ALL_NIBBLE_LSB
);
THIS^.testValueIsGreaterThan(
	valueToTest := THIS^.TOD_ALL_NIBBLE_MSB,
	lessValue := THIS^.TOD_ALL_NIBBLE_LSB
);
THIS^.testValueIsGreaterThan(
	valueToTest := THIS^.TOD_ALL_NIBBLE_LSB,
	lessValue := THIS^.TOD_ALL_NIBBLE_MSB
);
THIS^.testValueIsGreaterThan(
	valueToTest := THIS^.TOD_LSB_ONLY,
	lessValue := THIS^.TOD_MSB_ONLY
);
THIS^.testValueIsGreaterThan(
	valueToTest := THIS^.TOD_MSB_ONLY,
	lessValue := THIS^.TOD_MSB_ONLY
);
THIS^.testValueIsGreaterThan(
	valueToTest := THIS^.TOD_MSB_ONLY,
	lessValue := THIS^.TOD_LSB_ONLY
);
THIS^.testValueIsGreaterThan(
	valueToTest := THIS^.TOD_LSB_IS_UNSET,
	lessValue := THIS^.TOD_MAX
);
THIS^.testValueIsGreaterThan(
	valueToTest := THIS^.TOD_MAX,
	lessValue := THIS^.TOD_LSB_IS_UNSET
);
TcUnit.TEST_FINISHED();
END_METHOD

(*

short summary
==================
This test method tests ``assert.dateAndTime.simple.timeOfDay.valueIsInRangeOf``
method of CNM_AssertionInterfaceLib library with various inputs

.. <legal notes>

legal notes
=================
| SPDX-FileCopyrightText: © 2022 ekvip automation GmbH <info@ekvip.de>
| SPDX-License-Identifier: Apache-2.0
| For details check: Apache-2.0_

.. _Apache-2.0: https://www.apache.org/licenses/LICENSE-2.0

.. </legal notes>

*)

METHOD runValueIsInRangeOfTests
RETURN (NOT TcUnit.TEST_ORDERED(THIS^.getTestNameFor('valueIsInRangeOf')));

THIS^.testValueIsInRangeOf(
	lowerLimit := THIS^.TOD_MIN,
	valueToTest := THIS^.TOD_MAX,
	upperLimit	:= THIS^.TOD_MAX
);
THIS^.testValueIsInRangeOf(
	lowerLimit := THIS^.TOD_MIN,
	valueToTest := THIS^.TOD_MIN,
	upperLimit	:= THIS^.TOD_MAX
);
THIS^.testValueIsInRangeOf(
	lowerLimit := THIS^.TOD_MAX,
	valueToTest := THIS^.TOD_MAX,
	upperLimit	:= THIS^.TOD_MIN
);
THIS^.testValueIsInRangeOf(
	lowerLimit := THIS^.TOD_MAX,
	valueToTest := THIS^.TOD_MIN,
	upperLimit	:= THIS^.TOD_MIN
);
THIS^.testValueIsInRangeOf(
	lowerLimit := THIS^.TOD_LSB_IS_UNSET,
	valueToTest := THIS^.TOD_MIN,
	upperLimit	:= THIS^.TOD_MAX
);
THIS^.testValueIsInRangeOf(
	lowerLimit := THIS^.TOD_MIN,
	valueToTest := THIS^.TOD_LSB_IS_UNSET,
	upperLimit	:= THIS^.TOD_MAX
);
THIS^.testValueIsInRangeOf(
	lowerLimit := THIS^.TOD_LSB_IS_UNSET,
	valueToTest := THIS^.TOD_LSB_IS_UNSET,
	upperLimit	:= THIS^.TOD_LSB_IS_UNSET
);
THIS^.testValueIsInRangeOf(
	lowerLimit := THIS^.TOD_ALL_NIBBLE_LSB,
	valueToTest := THIS^.TOD_LSB_IS_UNSET,
	upperLimit	:= THIS^.TOD_ALL_NIBBLE_MSB
);
THIS^.testValueIsInRangeOf(
	lowerLimit := THIS^.TOD_LSB_IS_UNSET,
	valueToTest := THIS^.TOD_ALL_NIBBLE_LSB,
	upperLimit	:= THIS^.TOD_ALL_NIBBLE_MSB
);
THIS^.testValueIsInRangeOf(
	lowerLimit := THIS^.TOD_LSB_ONLY,
	valueToTest := THIS^.TOD_WITHOUT_MSB,
	upperLimit	:= THIS^.TOD_MSB_ONLY
);
THIS^.testValueIsInRangeOf(
	lowerLimit := THIS^.TOD_WITHOUT_MSB,
	valueToTest := THIS^.TOD_LSB_ONLY,
	upperLimit	:= THIS^.TOD_MSB_ONLY
);
THIS^.testValueIsInRangeOf(
	lowerLimit := THIS^.TOD_WITHOUT_NIBBLE_MSB,
	valueToTest := THIS^.TOD_MAX,
	upperLimit	:= THIS^.TOD_ALL_NIBBLE_MSB
);
THIS^.testValueIsInRangeOf(
	lowerLimit := THIS^.TOD_WITHOUT_NIBBLE_MSB,
	valueToTest := THIS^.TOD_MIN,
	upperLimit	:= THIS^.TOD_ALL_NIBBLE_MSB
);
THIS^.testValueIsInRangeOf(
	lowerLimit := THIS^.TOD_WITHOUT_NIBBLE_MSB,
	valueToTest := THIS^.TOD_WITHOUT_NIBBLE_MSB,
	upperLimit	:= THIS^.TOD_ALL_NIBBLE_MSB
);
THIS^.testValueIsInRangeOf(
	lowerLimit := THIS^.TOD_WITHOUT_NIBBLE_MSB,
	valueToTest := THIS^.TOD_ALL_NIBBLE_MSB,
	upperLimit	:= THIS^.TOD_ALL_NIBBLE_MSB
);
TcUnit.TEST_FINISHED();
END_METHOD

(*

short summary
==================
This test method tests ``assert.dateAndTime.simple.timeOfDay.valueIsLessThan``
method of CNM_AssertionInterfaceLib library with various inputs

.. <legal notes>

legal notes
=================
| SPDX-FileCopyrightText: © 2022 ekvip automation GmbH <info@ekvip.de>
| SPDX-License-Identifier: Apache-2.0
| For details check: Apache-2.0_

.. _Apache-2.0: https://www.apache.org/licenses/LICENSE-2.0

.. </legal notes>

*)

METHOD runValueIsLessThanTests
RETURN (NOT TcUnit.TEST_ORDERED(THIS^.getTestNameFor('valueIsLessThan')));

THIS^.testValueIsLessThan(
	valueToTest := THIS^.TOD_MAX,
	greaterValue := THIS^.TOD_MAX
);
THIS^.testValueIsLessThan(
	valueToTest := THIS^.TOD_MIN,
	greaterValue := THIS^.TOD_MIN
);
THIS^.testValueIsLessThan(
	valueToTest := THIS^.TOD_MIN,
	greaterValue := THIS^.TOD_MAX
);
THIS^.testValueIsLessThan(
	valueToTest := THIS^.TOD_MAX,
	greaterValue := THIS^.TOD_MIN
);
THIS^.testValueIsLessThan(
	valueToTest := THIS^.TOD_ALL_NIBBLE_LSB,
	greaterValue := THIS^.TOD_ALL_NIBBLE_LSB
);
THIS^.testValueIsLessThan(
	valueToTest := THIS^.TOD_ALL_NIBBLE_MSB,
	greaterValue := THIS^.TOD_ALL_NIBBLE_LSB
);
THIS^.testValueIsLessThan(
	valueToTest := THIS^.TOD_ALL_NIBBLE_LSB,
	greaterValue := THIS^.TOD_ALL_NIBBLE_MSB
);
THIS^.testValueIsLessThan(
	valueToTest := THIS^.TOD_LSB_ONLY,
	greaterValue := THIS^.TOD_MSB_ONLY
);
THIS^.testValueIsLessThan(
	valueToTest := THIS^.TOD_MSB_ONLY,
	greaterValue := THIS^.TOD_MSB_ONLY
);
THIS^.testValueIsLessThan(
	valueToTest := THIS^.TOD_MSB_ONLY,
	greaterValue := THIS^.TOD_LSB_ONLY
);
THIS^.testValueIsLessThan(
	valueToTest := THIS^.TOD_LSB_IS_UNSET,
	greaterValue := THIS^.TOD_MAX
);
THIS^.testValueIsLessThan(
	valueToTest := THIS^.TOD_MAX,
	greaterValue := THIS^.TOD_LSB_IS_UNSET
);
TcUnit.TEST_FINISHED();
END_METHOD

(*

short summary
==================
This test method tests ``assert.dateAndTime.simple.timeOfDay.valueIsMax``
method of CNM_AssertionInterfaceLib library with various inputs

.. <legal notes>

legal notes
=================
| SPDX-FileCopyrightText: © 2022 ekvip automation GmbH <info@ekvip.de>
| SPDX-License-Identifier: Apache-2.0
| For details check: Apache-2.0_

.. _Apache-2.0: https://www.apache.org/licenses/LICENSE-2.0

.. </legal notes>

*)

METHOD runValueIsMaxTests
RETURN (NOT TcUnit.TEST_ORDERED(THIS^.getTestNameFor('valueIsMax')));

THIS^.testValueIsMax(
	valueToTest := THIS^.TOD_MAX,
	maximumValue := THIS^.TOD_MAX
);
THIS^.testValueIsMax(
	valueToTest := THIS^.TOD_MIN,
	maximumValue := THIS^.TOD_MIN
);
THIS^.testValueIsMax(
	valueToTest := THIS^.TOD_MIN,
	maximumValue := THIS^.TOD_MAX
);
THIS^.testValueIsMax(
	valueToTest := THIS^.TOD_MAX,
	maximumValue := THIS^.TOD_MIN
);
THIS^.testValueIsMax(
	valueToTest := THIS^.TOD_ALL_NIBBLE_LSB,
	maximumValue := THIS^.TOD_ALL_NIBBLE_LSB
);
THIS^.testValueIsMax(
	valueToTest := THIS^.TOD_ALL_NIBBLE_MSB,
	maximumValue := THIS^.TOD_ALL_NIBBLE_LSB
);
THIS^.testValueIsMax(
	valueToTest := THIS^.TOD_ALL_NIBBLE_LSB,
	maximumValue := THIS^.TOD_ALL_NIBBLE_MSB
);
THIS^.testValueIsMax(
	valueToTest := THIS^.TOD_LSB_ONLY,
	maximumValue := THIS^.TOD_MSB_ONLY
);
THIS^.testValueIsMax(
	valueToTest := THIS^.TOD_MSB_ONLY,
	maximumValue := THIS^.TOD_MSB_ONLY
);
THIS^.testValueIsMax(
	valueToTest := THIS^.TOD_MSB_ONLY,
	maximumValue := THIS^.TOD_LSB_ONLY
);
THIS^.testValueIsMax(
	valueToTest := THIS^.TOD_LSB_IS_UNSET,
	maximumValue := THIS^.TOD_MAX
);
THIS^.testValueIsMax(
	valueToTest := THIS^.TOD_MAX,
	maximumValue := THIS^.TOD_LSB_IS_UNSET
);
TcUnit.TEST_FINISHED();
END_METHOD

(*

short summary
==================
This test method tests ``assert.dateAndTime.simple.timeOfDay.valueIsMin``
method of CNM_AssertionInterfaceLib library with various inputs

.. <legal notes>

legal notes
=================
| SPDX-FileCopyrightText: © 2022 ekvip automation GmbH <info@ekvip.de>
| SPDX-License-Identifier: Apache-2.0
| For details check: Apache-2.0_

.. _Apache-2.0: https://www.apache.org/licenses/LICENSE-2.0

.. </legal notes>

*)

METHOD runValueIsMinTests
RETURN (NOT TcUnit.TEST_ORDERED(THIS^.getTestNameFor('valueIsMin')));

THIS^.testValueIsMin(
	valueToTest := THIS^.TOD_MAX,
	minimumValue := THIS^.TOD_MAX
);
THIS^.testValueIsMin(
	valueToTest := THIS^.TOD_MIN,
	minimumValue := THIS^.TOD_MIN
);
THIS^.testValueIsMin(
	valueToTest := THIS^.TOD_MIN,
	minimumValue := THIS^.TOD_MAX
);
THIS^.testValueIsMin(
	valueToTest := THIS^.TOD_MAX,
	minimumValue := THIS^.TOD_MIN
);
THIS^.testValueIsMin(
	valueToTest := THIS^.TOD_ALL_NIBBLE_LSB,
	minimumValue := THIS^.TOD_ALL_NIBBLE_LSB
);
THIS^.testValueIsMin(
	valueToTest := THIS^.TOD_ALL_NIBBLE_MSB,
	minimumValue := THIS^.TOD_ALL_NIBBLE_LSB
);
THIS^.testValueIsMin(
	valueToTest := THIS^.TOD_ALL_NIBBLE_LSB,
	minimumValue := THIS^.TOD_ALL_NIBBLE_MSB
);
THIS^.testValueIsMin(
	valueToTest := THIS^.TOD_LSB_ONLY,
	minimumValue := THIS^.TOD_MSB_ONLY
);
THIS^.testValueIsMin(
	valueToTest := THIS^.TOD_MSB_ONLY,
	minimumValue := THIS^.TOD_MSB_ONLY
);
THIS^.testValueIsMin(
	valueToTest := THIS^.TOD_MSB_ONLY,
	minimumValue := THIS^.TOD_LSB_ONLY
);
THIS^.testValueIsMin(
	valueToTest := THIS^.TOD_LSB_IS_UNSET,
	minimumValue := THIS^.TOD_MAX
);
THIS^.testValueIsMin(
	valueToTest := THIS^.TOD_MAX,
	minimumValue := THIS^.TOD_LSB_IS_UNSET
);
TcUnit.TEST_FINISHED();
END_METHOD

(*

short summary
==================
This test method tests ``assert.dateAndTime.simple.timeOfDay.valueIsNotEqualTo``
method of CNM_AssertionInterfaceLib library with various inputs

.. <legal notes>

legal notes
=================
| SPDX-FileCopyrightText: © 2022 ekvip automation GmbH <info@ekvip.de>
| SPDX-License-Identifier: Apache-2.0
| For details check: Apache-2.0_

.. _Apache-2.0: https://www.apache.org/licenses/LICENSE-2.0

.. </legal notes>

*)

METHOD runValueIsNotEqualToTests
RETURN (NOT TcUnit.TEST_ORDERED(THIS^.getTestNameFor('valueIsNotEqualTo')));

THIS^.testValueIsNotEqualTo(
	valueToTest := THIS^.TOD_MAX,
	unexpectedValue := THIS^.TOD_MAX
);
THIS^.testValueIsNotEqualTo(
	valueToTest := THIS^.TOD_MIN,
	unexpectedValue := THIS^.TOD_MIN
);
THIS^.testValueIsNotEqualTo(
	valueToTest := THIS^.TOD_MIN,
	unexpectedValue := THIS^.TOD_MAX
);
THIS^.testValueIsNotEqualTo(
	valueToTest := THIS^.TOD_MAX,
	unexpectedValue := THIS^.TOD_MIN
);
THIS^.testValueIsNotEqualTo(
	valueToTest := THIS^.TOD_ALL_NIBBLE_LSB,
	unexpectedValue := THIS^.TOD_ALL_NIBBLE_LSB
);
THIS^.testValueIsNotEqualTo(
	valueToTest := THIS^.TOD_LSB_ONLY,
	unexpectedValue := THIS^.TOD_MSB_ONLY
);
THIS^.testValueIsNotEqualTo(
	valueToTest := THIS^.TOD_MSB_ONLY,
	unexpectedValue := THIS^.TOD_MSB_ONLY
);
THIS^.testValueIsNotEqualTo(
	valueToTest := THIS^.TOD_MSB_ONLY,
	unexpectedValue := THIS^.TOD_LSB_ONLY
);

TcUnit.TEST_FINISHED();
END_METHOD

(*

short summary
==================
This test method tests ``assert.dateAndTime.simple.timeOfDay.valueIsEqualTo``
method of CNM_AssertionInterfaceLib library, 
it provides the possibility to handover test data via parameter 


.. <legal notes>

legal notes
=================
| SPDX-FileCopyrightText: © 2022 ekvip automation GmbH <info@ekvip.de>
| SPDX-License-Identifier: Apache-2.0
| For details check: Apache-2.0_

.. _Apache-2.0: https://www.apache.org/licenses/LICENSE-2.0

.. </legal notes>

parameters
==========

*)

METHOD testValueIsEqualTo 
VAR_INPUT
	(* for the test it's the parameter ``currentValue`` *)
	valueToTest	:TOD;
	(* for the test it's the parameter ``expectedValue`` *)
	expected	:TOD;
END_VAR
VAR
	(* just the expectation if the assertion to test must be worng or true *)
	assertionIsWrong		:BOOL;
	(* contains the format string for the test message *)
	message					:Tc2_System.T_MaxString;
	(* TwinCAT printf with the test message *)
	messageStringBuilder	:Tc2_Utilities.FB_FormatString;
	(* TOD value of ``currentValue`` as string *)
	currentValueAsString	:STRING(22);
	(* TOD value of ``expectedValue`` as string *)
	expectedValueAsString	:STRING(22);
END_VAR
THIS^.assertorContainer.resetAssertor();

assertionIsWrong := (valueToTest <> expected);
message := SEL(
	assertionIsWrong,
	'currentValue is %s expectedValue is %s assertion must be TRUE', 
	'currentValue is %s expectedValue is %s assertion must be FALSE'
);
currentValueAsString := TO_STRING(valueToTest);
expectedValueAsString := TO_STRING(expected);

messageStringBuilder(
	sFormat := message,
	arg1 := THIS^.AnyToArg(currentValueAsString),
	arg2 := THIS^.AnyToArg(expectedValueAsString)
);

THIS^.assertorContainer.assertor.assert.dateAndTime.simple.timeOfDay.valueIsEqualTo(
	currentValue	:= valueToTest,
	expectedValue	:= expected,
	message			:= ''
   );

THIS^.AssertEquals_BOOL(
	Expected 	:= assertionIsWrong,
	Actual 		:= THIS^.assertorContainer.wasAssertionWrong,
	Message 	:= messageStringBuilder.sOut
);
END_METHOD

(*

short summary
==================
This test method tests ``assert.dateAndTime.simple.timeOfDay.valueIsGreaterThan``
method of CNM_AssertionInterfaceLib library, 
it provides the possibility to handover test data via parameter 


.. <legal notes>

legal notes
=================
| SPDX-FileCopyrightText: © 2022 ekvip automation GmbH <info@ekvip.de>
| SPDX-License-Identifier: Apache-2.0
| For details check: Apache-2.0_

.. _Apache-2.0: https://www.apache.org/licenses/LICENSE-2.0

.. </legal notes>

parameters
==========

*)

METHOD testValueIsGreaterThan 
VAR_INPUT
	(* for the test it's the parameter ``currentValue`` *)
	valueToTest	:TOD;
	(* for the test it's the parameter ``lessValue`` *)
	lessValue	:TOD;
END_VAR
VAR
	(* just the expectation if the assertion to test must be worng or true *)
	assertionIsWrong		:BOOL;
	(* contains the format string for the test message *)
	message					:Tc2_System.T_MaxString;
	(* TwinCAT printf with the test message *)
	messageStringBuilder	:Tc2_Utilities.FB_FormatString;
	(* TOD value of ``currentValue`` as string *)
	currentValueAsString	:STRING(22);
	(* TOD value of ``lessValue`` as string *)
	lessValueAsString		:STRING(22);
END_VAR
THIS^.assertorContainer.resetAssertor();

assertionIsWrong := (valueToTest <= lessValue);
message := SEL(
	assertionIsWrong,
	'currentValue is %s lessValue is %s assertion must be TRUE', 
	'currentValue is %s lessValue is %s assertion must be FALSE'
);
currentValueAsString := TO_STRING(valueToTest);
lessValueAsString := TO_STRING(lessValue);

messageStringBuilder(
	sFormat := message,
	arg1 := THIS^.AnyToArg(currentValueAsString),
	arg2 := THIS^.AnyToArg(lessValueAsString)
);

THIS^.assertorContainer.assertor.assert.dateAndTime.simple.timeOfDay.valueIsGreaterThan(
	currentValue	:= valueToTest,
	lessValue		:= lessValue,
	message			:= ''
   );

THIS^.AssertEquals_BOOL(
	Expected 	:= assertionIsWrong,
	Actual 		:= THIS^.assertorContainer.wasAssertionWrong,
	Message 	:= messageStringBuilder.sOut
);
END_METHOD

(*

short summary
==================
This test method tests ``assert.dateAndTime.simple.timeOfDay.valueIsInRangeOf``
method of CNM_AssertionInterfaceLib library, 
it provides the possibility to handover test data via parameter 


.. <legal notes>

legal notes
=================
| SPDX-FileCopyrightText: © 2022 ekvip automation GmbH <info@ekvip.de>
| SPDX-License-Identifier: Apache-2.0
| For details check: Apache-2.0_

.. _Apache-2.0: https://www.apache.org/licenses/LICENSE-2.0

.. </legal notes>

parameters
==========

*)

METHOD testValueIsInRangeOf 
VAR_INPUT
	(* for the test it's the parameter ``lowerLimit`` *)
	lowerLimit	:TOD;
	(* for the test it's the parameter ``currentValue`` *)
	valueToTest	:TOD;
	(* for the test it's the parameter ``upperLimit`` *)
	upperLimit	:TOD;
END_VAR
VAR
	(* just the expectation if the assertion to test must be worng or true *)
	assertionIsWrong		:BOOL;
	(* contains the format string for the test message *)
	message					:Tc2_System.T_MaxString;
	(* TwinCAT printf with the test message *)
	messageStringBuilder	:Tc2_Utilities.FB_FormatString;
	(* TOD value of ``lowerLimit`` as string *)
	lowerLimitAsString		:STRING(22);
	(* TOD value of ``currentValue`` as string *)
	currentValueAsString	:STRING(22);
	(* TOD value of ``upperLimit`` as string *)
	upperLimitAsString		:STRING(22);
END_VAR
THIS^.assertorContainer.resetAssertor();

assertionIsWrong := ((valueToTest < lowerLimit) OR (valueToTest > upperLimit));
message := SEL(
	assertionIsWrong,
	'lowerLimit is %s currentValue is %s upperLimit is %s assertion must be TRUE', 
	'lowerLimit is %s currentValue is %s upperLimit is %s assertion must be FALSE'
);
lowerLimitAsString		:= TO_STRING(lowerLimit);
currentValueAsString	:= TO_STRING(valueToTest);
upperLimitAsString		:= TO_STRING(upperLimit);

messageStringBuilder(
	sFormat := message,
	arg1 := THIS^.AnyToArg(lowerLimitAsString),
	arg2 := THIS^.AnyToArg(currentValueAsString),
	arg3 := THIS^.AnyToArg(upperLimitAsString)
);

THIS^.assertorContainer.assertor.assert.dateAndTime.simple.timeOfDay.valueIsInRangeOf(
	lowerLimit		:= lowerLimit,
	currentValue	:= valueToTest,
	upperLimit		:= upperLimit,
	message			:= ''
   );

THIS^.AssertEquals_BOOL(
	Expected 	:= assertionIsWrong,
	Actual 		:= THIS^.assertorContainer.wasAssertionWrong,
	Message 	:= messageStringBuilder.sOut
);
END_METHOD

(*

short summary
==================
This test method tests ``assert.dateAndTime.simple.timeOfDay.valueIsLessThan``
method of CNM_AssertionInterfaceLib library, 
it provides the possibility to handover test data via parameter 


.. <legal notes>

legal notes
=================
| SPDX-FileCopyrightText: © 2022 ekvip automation GmbH <info@ekvip.de>
| SPDX-License-Identifier: Apache-2.0
| For details check: Apache-2.0_

.. _Apache-2.0: https://www.apache.org/licenses/LICENSE-2.0

.. </legal notes>

parameters
==========

*)

METHOD testValueIsLessThan 
VAR_INPUT
	(* for the test it's the parameter ``currentValue`` *)
	valueToTest		:TOD;
	(* for the test it's the parameter ``greaterValue`` *)
	greaterValue	:TOD;
END_VAR
VAR
	(* just the expectation if the assertion to test must be worng or true *)
	assertionIsWrong		:BOOL;
	(* contains the format string for the test message *)
	message					:Tc2_System.T_MaxString;
	(* TwinCAT printf with the test message *)
	messageStringBuilder	:Tc2_Utilities.FB_FormatString;
	(* TOD value of ``currentValue`` as string *)
	currentValueAsString	:STRING(22);
	(* TOD value of ``greaterValue`` as string *)
	greaterValueAsString	:STRING(22);
END_VAR
THIS^.assertorContainer.resetAssertor();

assertionIsWrong := (valueToTest >= greaterValue);
message := SEL(
	assertionIsWrong,
	'currentValue is %s greaterValue is %s assertion must be TRUE', 
	'currentValue is %s greaterValue is %s assertion must be FALSE'
);
currentValueAsString := TO_STRING(valueToTest);
greaterValueAsString := TO_STRING(greaterValue);

messageStringBuilder(
	sFormat := message,
	arg1 := THIS^.AnyToArg(currentValueAsString),
	arg2 := THIS^.AnyToArg(greaterValueAsString)
);

THIS^.assertorContainer.assertor.assert.dateAndTime.simple.timeOfDay.valueIsLessThan(
	currentValue	:= valueToTest,
	greaterValue	:= greaterValue,
	message			:= ''
   );

THIS^.AssertEquals_BOOL(
	Expected 	:= assertionIsWrong,
	Actual 		:= THIS^.assertorContainer.wasAssertionWrong,
	Message 	:= messageStringBuilder.sOut
);
END_METHOD

(*

short summary
==================
This test method tests ``assert.dateAndTime.simple.timeOfDay.valueIsMax``
method of CNM_AssertionInterfaceLib library, 
it provides the possibility to handover test data via parameter 


.. <legal notes>

legal notes
=================
| SPDX-FileCopyrightText: © 2022 ekvip automation GmbH <info@ekvip.de>
| SPDX-License-Identifier: Apache-2.0
| For details check: Apache-2.0_

.. _Apache-2.0: https://www.apache.org/licenses/LICENSE-2.0

.. </legal notes>

parameters
==========

*)

METHOD testValueIsMax 
VAR_INPUT
	(* for the test it's the parameter ``currentValue`` *)
	valueToTest		:TOD;
	(* for the test it's the parameter ``greaterValue`` *)
	maximumValue	:TOD;
END_VAR
VAR
	(* just the expectation if the assertion to test must be worng or true *)
	assertionIsWrong		:BOOL;
	(* contains the format string for the test message *)
	message					:Tc2_System.T_MaxString;
	(* TwinCAT printf with the test message *)
	messageStringBuilder	:Tc2_Utilities.FB_FormatString;
	(* TOD value of ``currentValue`` as string *)
	currentValueAsString	:STRING(22);
	(* TOD value of ``maximumValue`` as string *)
	maximumValueAsString	:STRING(22);
END_VAR
THIS^.assertorContainer.resetAssertor();

assertionIsWrong := (valueToTest > maximumValue);
message := SEL(
	assertionIsWrong,
	'currentValue is %s maximumValue is %s assertion must be TRUE', 
	'currentValue is %s maximumValue is %s assertion must be FALSE'
);
currentValueAsString := TO_STRING(valueToTest);
maximumValueAsString := TO_STRING(maximumValue);

messageStringBuilder(
	sFormat := message,
	arg1 := THIS^.AnyToArg(currentValueAsString),
	arg2 := THIS^.AnyToArg(maximumValueAsString)
);

THIS^.assertorContainer.assertor.assert.dateAndTime.simple.timeOfDay.valueIsMax(
	currentValue	:= valueToTest,
	maximumValue	:= maximumValue,
	message			:= ''
   );

THIS^.AssertEquals_BOOL(
	Expected 	:= assertionIsWrong,
	Actual 		:= THIS^.assertorContainer.wasAssertionWrong,
	Message 	:= messageStringBuilder.sOut
);
END_METHOD

(*

short summary
==================
This test method tests ``assert.dateAndTime.simple.timeOfDay.valueIsMin``
method of CNM_AssertionInterfaceLib library, 
it provides the possibility to handover test data via parameter 


.. <legal notes>

legal notes
=================
| SPDX-FileCopyrightText: © 2022 ekvip automation GmbH <info@ekvip.de>
| SPDX-License-Identifier: Apache-2.0
| For details check: Apache-2.0_

.. _Apache-2.0: https://www.apache.org/licenses/LICENSE-2.0

.. </legal notes>

parameters
==========

*)

METHOD testValueIsMin 
VAR_INPUT
	(* for the test it's the parameter ``currentValue`` *)
	valueToTest		:TOD;
	(* for the test it's the parameter ``greaterValue`` *)
	minimumValue	:TOD;
END_VAR
VAR
	(* just the expectation if the assertion to test must be worng or true *)
	assertionIsWrong		:BOOL;
	(* contains the format string for the test message *)
	message					:Tc2_System.T_MaxString;
	(* TwinCAT printf with the test message *)
	messageStringBuilder	:Tc2_Utilities.FB_FormatString;
	(* TOD value of ``currentValue`` as string *)
	currentValueAsString	:STRING(22);
	(* TOD value of ``minimumValue`` as string *)
	minimumValueAsString	:STRING(22);
END_VAR
THIS^.assertorContainer.resetAssertor();

assertionIsWrong := (valueToTest < minimumValue);
message := SEL(
	assertionIsWrong,
	'currentValue is %s minimumValue is %s assertion must be TRUE', 
	'currentValue is %s minimumValue is %s assertion must be FALSE'
);
currentValueAsString := TO_STRING(valueToTest);
minimumValueAsString := TO_STRING(minimumValue);

messageStringBuilder(
	sFormat := message,
	arg1 := THIS^.AnyToArg(currentValueAsString),
	arg2 := THIS^.AnyToArg(minimumValueAsString)
);

THIS^.assertorContainer.assertor.assert.dateAndTime.simple.timeOfDay.valueIsMin(
	currentValue	:= valueToTest,
	minimumValue	:= minimumValue,
	message			:= ''
   );

THIS^.AssertEquals_BOOL(
	Expected 	:= assertionIsWrong,
	Actual 		:= THIS^.assertorContainer.wasAssertionWrong,
	Message 	:= messageStringBuilder.sOut
);
END_METHOD

(*

short summary
==================
This test method tests ``assert.dateAndTime.simple.timeOfDay.valueIsNotEqualTo``
method of CNM_AssertionInterfaceLib library, 
it provides the possibility to handover test data via parameter 


.. <legal notes>

legal notes
=================
| SPDX-FileCopyrightText: © 2022 ekvip automation GmbH <info@ekvip.de>
| SPDX-License-Identifier: Apache-2.0
| For details check: Apache-2.0_

.. _Apache-2.0: https://www.apache.org/licenses/LICENSE-2.0

.. </legal notes>

parameters
==========

*)

METHOD testValueIsNotEqualTo 
VAR_INPUT
	(* for the test it's the parameter ``currentValue`` *)
	valueToTest		:TOD;
	(* for the test it's the parameter ``unexpectedValue`` *)
	unexpectedValue	:TOD;
END_VAR
VAR
	(* just the expectation if the assertion to test must be worng or true *)
	assertionIsWrong		:BOOL;
	(* contains the format string for the test message *)
	message					:Tc2_System.T_MaxString;
	(* TwinCAT printf with the test message *)
	messageStringBuilder	:Tc2_Utilities.FB_FormatString;
	(* TOD value of ``currentValue`` as string *)
	currentValueAsString	:STRING(22);
	(* TOD value of ``unexpectedValue`` as string *)
	unexpectedValueAsString	:STRING(22);
END_VAR
THIS^.assertorContainer.resetAssertor();

assertionIsWrong := (valueToTest = unexpectedValue);
message := SEL(
	assertionIsWrong,
	'currentValue is %s expectedValue is %s assertion must be TRUE', 
	'currentValue is %s expectedValue is %s assertion must be FALSE'
);
currentValueAsString := TO_STRING(valueToTest);
unexpectedValueAsString := TO_STRING(unexpectedValue);

messageStringBuilder(
	sFormat := message,
	arg1 := THIS^.AnyToArg(currentValueAsString),
	arg2 := THIS^.AnyToArg(unexpectedValueAsString)
);

THIS^.assertorContainer.assertor.assert.dateAndTime.simple.timeOfDay.valueIsNotEqualTo(
	currentValue	:= valueToTest,
	unexpectedValue	:= unexpectedValue,
	message			:= ''
   );

THIS^.AssertEquals_BOOL(
	Expected 	:= assertionIsWrong,
	Actual 		:= THIS^.assertorContainer.wasAssertionWrong,
	Message 	:= messageStringBuilder.sOut
);
END_METHOD

END_FUNCTION_BLOCK

// ---- AssertionTester/AssertionTests/FloatAssertions/classes/RealAssertionTests.TcPOU
(*

short summary
==================
This class tests all methods of REAL assertions
with various combinations of inputs and checks expected 
outputs are satisfied or not

.. <legal notes>

legal notes
=================
| SPDX-FileCopyrightText: © 2022 ekvip automation GmbH <info@ekvip.de>
| SPDX-License-Identifier: Apache-2.0
| For details check: Apache-2.0_

.. _Apache-2.0: https://www.apache.org/licenses/LICENSE-2.0

.. </legal notes>

methods and properties
======================

*)


FUNCTION_BLOCK RealAssertionTests EXTENDS AbstractAssertorTest
VAR
	(* not a number *)
	NAN							:REAL;
	(* infinity *)
	INF							:REAL;
	(* -infinity *)
	MINUS_INF					:REAL;
	(* -0.0 (MSB is set only) *)
	MINUS_ZERO					:REAL;
	(* minimum subnormal value (all fraction bits and MSB set only) *)
	MIN_SUBNORMAL				:REAL;
	(* maximum subnormal value (all fraction bits are set only) *)
	MAX_SUBNORMAL				:REAL;
	(* smallest positive subnormal value (LSB set only)*)
	SMALLEST_POSITIVE_SUBNORMAL	:REAL;
	(* smallest negative subnormal value (LSB and MSB set only)*)
	SMALLEST_NEGATIVE_SUBNORMAL	:REAL;
END_VAR
VAR CONSTANT
	(* prefix to unify the test names *)
	TEST_NAME_PREFIX					:STRING := 'assert.float.single.';
	(* max value of real *)
	MAX_NON_SPECIAL						:REAL := 3.402823E+38;
	(* min value of real *)
	MIN_NON_SPECIAL						:REAL := -3.402823E+38;
	(* 0.0 *)
	ZERO								:REAL := 0.0;
	(* 1% *)
	ONE_PERCENT							:REAL := 0.01;
	(* 1‰ *)
	ONE_PERMILLE						:REAL := 0.001;
	(* bit number of the sign bit *)
	SIGN								:USINT := 31;
	(* binary value of 0.0 *)
	BINARY_ZERO							:DWORD := 16#0000_0000;
	(* binary value of -0.0 *)
	BINARY_MINUS_ZERO					:DWORD := 16#8000_0000;
	(* binary value of inf *)
	BINARY_INFINITY						:DWORD := 16#7F80_0000;
	(* binary value of -inf *)
	BINARY_NEGATIVE_INFINITY			:DWORD := 16#FF80_0000;
	(* mask to filter the exponent of the number *)
	MASK_FOR_EXPONENT					:DWORD := 16#7F80_0000;
	(* minimum denormalized number *)
	BINARY_MIN_SUBNORMAL				:DWORD := 16#807F_FFFF;
	(* maximum denormalized number*)
	BINARY_MAX_SUBNORMAL				:DWORD := 16#007F_FFFF;
	(* smallest positive denormalizied number greater than zero *)
	BINARY_SMALLEST_POSITIVE_SUBNORMAL	:DWORD := 16#0000_0001;
	(* smallest negative denormalizied number greater than minus zero *)
	BINARY_SMALLEST_NEGATIVE_SUBNORMAL	:DWORD := 16#8000_0001;
	(* smallest positive signaling NaN *)
	BINARY_POSITIVE_SIGNALING_NAN		:DWORD := 16#7F80_0001;
END_VAR

THIS^.runValueIsEqualToTests();
THIS^.runValueIsGreaterThanTests();
THIS^.runValueIsInRangeOfTests();
THIS^.runValueIsLessThanTests();
THIS^.runValueIsMaxTests();
THIS^.runValueIsMinTests();
THIS^.runValueIsNotEqualToTests();
THIS^.runValueIsANumberTests();
THIS^.runValueIsFiniteTests();
THIS^.runValueIsInfiniteTests();
THIS^.runValueIsNaNTests();
THIS^.runValueIsNegativeTests();
THIS^.runValueIsPositiveTests();
THIS^.runValueIsNegativeInfiniteTests();
THIS^.runValueIsPositiveInfiniteTests();
THIS^.runValueIsNegativeZeroTests();
THIS^.runValueIsPositiveZeroTests();
THIS^.runValueIsNormalTests();
THIS^.runValueIsNotNegativeInfiniteTests();
THIS^.runValueIsNotPositiveInfiniteTests();
THIS^.runValueIsNotSpecialTests();
THIS^.runValueIsSpecialTests();
THIS^.runValueIsSubnormalTests();

(*

short summary
=============
It attaches the container with the class to test
and it sets the special numbers from `IEEE 754`_ standard

.. _IEEE 754: https://en.wikipedia.org/wiki/IEEE_754

legal notes
=================
| SPDX-FileCopyrightText: © 2023 ekvip automation GmbH <info@ekvip.de>
| SPDX-License-Identifier: Apache-2.0
| For details check: Apache-2.0_

.. _Apache-2.0: https://www.apache.org/licenses/LICENSE-2.0

.. </legal notes>

parameters
==========

*)

METHOD FB_init :BOOL
VAR_INPUT
	(* if TRUE, the retain variables are initialized (warm start / cold start) *)
    bInitRetains	:BOOL;
	(* if TRUE, the instance afterwards gets moved into the copy code (online change) *)
    bInCopyCode		:BOOL;
	(* container with the class to test *)
	classToBeTested :IAssertorContainer;
END_VAR
VAR
	{attribute 'hide'}
	newHashstate3		:CNM_AbstractObject.Hashcode;
	{attribute 'hide'}
	carzyNumberPointer	:POINTER TO DWORD;	
END_VAR
VAR CONSTANT
	{attribute 'hide'}
	NUMBER_OF_LEFT_SHIFTS		:UINT	:= 17;
	{attribute 'hide'}
	NUMBER_OF_LEFT_ROTATIONS	:UINT   := 45;
END_VAR
carzyNumberPointer := ADR(THIS^.NAN);
carzyNumberPointer^ := THIS^.BINARY_POSITIVE_SIGNALING_NAN;

carzyNumberPointer := ADR(THIS^.INF);
carzyNumberPointer^ := THIS^.BINARY_INFINITY;

carzyNumberPointer := ADR(THIS^.MINUS_INF);
carzyNumberPointer^ := THIS^.BINARY_NEGATIVE_INFINITY;

carzyNumberPointer := ADR(THIS^.MINUS_ZERO);
carzyNumberPointer^ := THIS^.BINARY_MINUS_ZERO;

carzyNumberPointer := ADR(THIS^.MIN_SUBNORMAL);
carzyNumberPointer^ := THIS^.BINARY_MIN_SUBNORMAL; 

carzyNumberPointer := ADR(THIS^.MAX_SUBNORMAL);
carzyNumberPointer^ := THIS^.BINARY_MAX_SUBNORMAL; 

carzyNumberPointer := ADR(THIS^.SMALLEST_POSITIVE_SUBNORMAL);
carzyNumberPointer^ := THIS^.BINARY_SMALLEST_POSITIVE_SUBNORMAL; 

carzyNumberPointer := ADR(THIS^.SMALLEST_NEGATIVE_SUBNORMAL);
carzyNumberPointer^ := THIS^.BINARY_SMALLEST_NEGATIVE_SUBNORMAL;
END_METHOD

(*

short summary
==================
This test method is a helper function to create a unified test name

.. <legal notes>

legal notes
=================
| SPDX-FileCopyrightText: © 2022 ekvip automation GmbH <info@ekvip.de>
| SPDX-License-Identifier: Apache-2.0
| For details check: Apache-2.0_

.. _Apache-2.0: https://www.apache.org/licenses/LICENSE-2.0

.. </legal notes>

parameters
==========

*)

METHOD PROTECTED getTestNameFor :Tc2_System.T_MaxString
VAR_INPUT
	(* name of the method to test, to create a unified test name *)
	nameOfMethodToTest	:Tc2_System.T_MaxString;
END_VAR
getTestNameFor := Tc2_Standard.CONCAT(THIS^.TEST_NAME_PREFIX, nameOfMethodToTest);
END_METHOD

(*

short summary
==================
This test method tests ``assert.float.single.valueIsANumber``
method of CNM_AssertionInterfaceLib library with various inputs

.. <legal notes>

legal notes
=================
| SPDX-FileCopyrightText: © 2022 ekvip automation GmbH <info@ekvip.de>
| SPDX-License-Identifier: Apache-2.0
| For details check: Apache-2.0_

.. _Apache-2.0: https://www.apache.org/licenses/LICENSE-2.0

.. </legal notes>

*)

METHOD runValueIsANumberTests
RETURN (NOT TcUnit.TEST_ORDERED(THIS^.getTestNameFor('valueIsANumber')));

THIS^.testValueIsANumber(THIS^.NAN);
THIS^.testValueIsANumber(THIS^.INF);
THIS^.testValueIsANumber(THIS^.MINUS_INF);
THIS^.testValueIsANumber(THIS^.MAX_NON_SPECIAL);
THIS^.testValueIsANumber(THIS^.MIN_NON_SPECIAL);
THIS^.testValueIsANumber(THIS^.ZERO);
THIS^.testValueIsANumber(THIS^.MINUS_ZERO);
THIS^.testValueIsANumber(THIS^.MAX_SUBNORMAL);
THIS^.testValueIsANumber(THIS^.MIN_SUBNORMAL);
THIS^.testValueIsANumber(THIS^.SMALLEST_NEGATIVE_SUBNORMAL);
THIS^.testValueIsANumber(THIS^.SMALLEST_POSITIVE_SUBNORMAL);
THIS^.testValueIsANumber(THIS^.ONE_PERCENT);
THIS^.testValueIsANumber(THIS^.ONE_PERMILLE);
THIS^.testValueIsANumber(THIS^.ONE_PERCENT * -1.0);
THIS^.testValueIsANumber(THIS^.ONE_PERMILLE * -1.0);

TcUnit.TEST_FINISHED();
END_METHOD

(*

short summary
==================
This test method tests ``assert.float.single.valueIsEqualTo``
method of CNM_AssertionInterfaceLib library with various inputs

.. <legal notes>

legal notes
=================
| SPDX-FileCopyrightText: © 2022 ekvip automation GmbH <info@ekvip.de>
| SPDX-License-Identifier: Apache-2.0
| For details check: Apache-2.0_

.. _Apache-2.0: https://www.apache.org/licenses/LICENSE-2.0

.. </legal notes>

*)

METHOD runValueIsEqualToTests
RETURN (NOT TcUnit.TEST_ORDERED(THIS^.getTestNameFor('valueIsEqualTo')));

THIS^.testValueIsEqualTo(
	valueToTest := THIS^.NAN,
	expected := THIS^.ONE_PERCENT,
	tolerance := THIS^.ONE_PERMILLE
);

THIS^.testValueIsEqualTo(
	valueToTest := THIS^.ONE_PERCENT,
	expected := THIS^.NAN,
	tolerance := THIS^.ONE_PERMILLE
);

THIS^.testValueIsEqualTo(
	valueToTest := THIS^.ONE_PERCENT,
	expected := THIS^.ONE_PERCENT,
	tolerance := THIS^.NAN
);

THIS^.testValueIsEqualTo(
	valueToTest := THIS^.NAN,
	expected := THIS^.NAN,
	tolerance := THIS^.ONE_PERCENT
);

THIS^.testValueIsEqualTo(
	valueToTest := THIS^.NAN,
	expected := THIS^.NAN,
	tolerance := THIS^.NAN
);

THIS^.testValueIsEqualTo(
	valueToTest := THIS^.INF,
	expected := THIS^.ONE_PERCENT,
	tolerance := THIS^.ONE_PERMILLE
);

THIS^.testValueIsEqualTo(
	valueToTest := THIS^.ONE_PERCENT,
	expected := THIS^.INF,
	tolerance := THIS^.ONE_PERMILLE
);

THIS^.testValueIsEqualTo(
	valueToTest := THIS^.ONE_PERCENT,
	expected := THIS^.ONE_PERCENT,
	tolerance := THIS^.INF
);

THIS^.testValueIsEqualTo(
	valueToTest := THIS^.INF,
	expected := THIS^.INF,
	tolerance := THIS^.ONE_PERCENT
);

THIS^.testValueIsEqualTo(
	valueToTest := THIS^.INF,
	expected := THIS^.INF,
	tolerance := THIS^.INF
);

THIS^.testValueIsEqualTo(
	valueToTest := THIS^.INF,
	expected := THIS^.MINUS_INF,
	tolerance := THIS^.INF
);

THIS^.testValueIsEqualTo(
	valueToTest := THIS^.MINUS_INF,
	expected := THIS^.ONE_PERCENT,
	tolerance := THIS^.ONE_PERMILLE
);

THIS^.testValueIsEqualTo(
	valueToTest := THIS^.ONE_PERCENT,
	expected := THIS^.MINUS_INF,
	tolerance := THIS^.ONE_PERMILLE
);

